REGION Network 33: RINSE-2_CLEANING_TIME_(PBFV-1,PBFV-17,PZDV-1,F-PUMP,PBFV-3,PBFV-4,PBFV-8,CIP-IN)
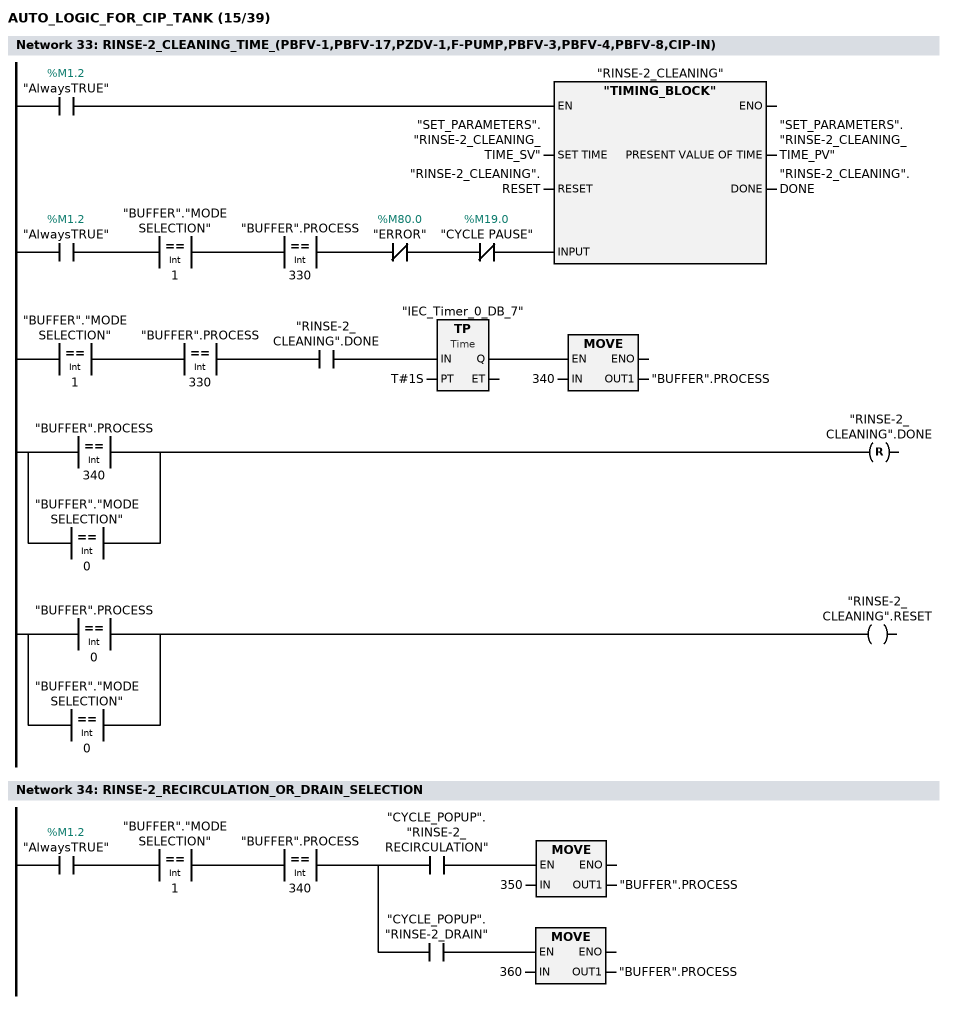
   RUNG wire#powerrail
      Contact( "AlwaysTRUE" )
      "RINSE-2_CLEANING"(INPUT := wire#w1, "SET TIME" := "SET_PARAMETERS"."RINSE-2_CLEANING_TIME_SV", RESET := "RINSE-2_CLEANING".RESET, "PRESENT VALUE OF TIME" => "SET_PARAMETERS"."RINSE-2_CLEANING_TIME_PV", DONE => "RINSE-2_CLEANING".DONE)
   END_RUNG
   RUNG wire#powerrail
      Contact( "AlwaysTRUE" )
      { S7_Templates := "SrcType := Int" } EQ_Contact(in1 := "BUFFER"."MODE SELECTION", in2 := 1)
      { S7_Templates := "SrcType := Int" } EQ_Contact(in1 := "BUFFER".PROCESS, in2 := 330)
      I_Contact( "ERROR" )
      I_Contact( "CYCLE PAUSE" )
   END_RUNG wire#w1
   RUNG wire#powerrail
      { S7_Templates := "SrcType := Int" } EQ_Contact(in1 := "BUFFER"."MODE SELECTION", in2 := 1)
      { S7_Templates := "SrcType := Int" } EQ_Contact(in1 := "BUFFER".PROCESS, in2 := 330)
      Contact( "RINSE-2_CLEANING".DONE )
      { S7_Templates := "time_type := Time" } "IEC_Timer_0_DB_7".TP(pt := T#1S, et =>)
      Move(in := 340, out1 => "BUFFER".PROCESS)
   END_RUNG
   RUNG wire#powerrail
      { S7_Templates := "SrcType := Int" } EQ_Contact(in1 := "BUFFER".PROCESS, in2 := 340)
      wire#w2
      R_Coil( "RINSE-2_CLEANING".DONE )
   END_RUNG
   RUNG wire#powerrail
      { S7_Templates := "SrcType := Int" } EQ_Contact(in1 := "BUFFER"."MODE SELECTION", in2 := 0)
   END_RUNG wire#w2
   RUNG wire#powerrail
      { S7_Templates := "SrcType := Int" } EQ_Contact(in1 := "BUFFER".PROCESS, in2 := 0)
      wire#w3
      Coil( "RINSE-2_CLEANING".RESET )
   END_RUNG
   RUNG wire#powerrail
      { S7_Templates := "SrcType := Int" } EQ_Contact(in1 := "BUFFER"."MODE SELECTION", in2 := 0)
   END_RUNG wire#w3
   // the same network as SCL:
   IF "AlwaysTRUE" THEN
       "RINSE-2_CLEANING"("SET TIME" := "SET_PARAMETERS"."RINSE-2_CLEANING_TIME_SV",   // "TIMING_BLOCK"
                          RESET := "RINSE-2_CLEANING".RESET,
                          INPUT := "AlwaysTRUE" AND ("BUFFER"."MODE SELECTION" = 1) AND ("BUFFER".PROCESS = 330) AND NOT "ERROR" AND NOT "CYCLE PAUSE",
                          "PRESENT VALUE OF TIME" => "SET_PARAMETERS"."RINSE-2_CLEANING_TIME_PV",
                          DONE => "RINSE-2_CLEANING".DONE);
   END_IF;
   "IEC_Timer_0_DB_7".TP(IN := ("BUFFER"."MODE SELECTION" = 1) AND ("BUFFER".PROCESS = 330) AND "RINSE-2_CLEANING".DONE,
                         PT := T#1S);
   IF "IEC_Timer_0_DB_7".Q THEN "BUFFER".PROCESS := 340; END_IF;
   IF ("BUFFER".PROCESS = 340) OR ("BUFFER"."MODE SELECTION" = 0) THEN
       "RINSE-2_CLEANING".DONE := FALSE;
   END_IF;
   "RINSE-2_CLEANING".RESET := ("BUFFER".PROCESS = 0) OR ("BUFFER"."MODE SELECTION" = 0);
END_REGION

REGION Network 34: RINSE-2_RECIRCULATION_OR_DRAIN_SELECTION
   RUNG wire#powerrail
      Contact( "AlwaysTRUE" )
      { S7_Templates := "SrcType := Int" } EQ_Contact(in1 := "BUFFER"."MODE SELECTION", in2 := 1)
      { S7_Templates := "SrcType := Int" } EQ_Contact(in1 := "BUFFER".PROCESS, in2 := 340)
      wire#w1
      Contact( "CYCLE_POPUP"."RINSE-2_RECIRCULATION" )
      Move(in := 350, out1 => "BUFFER".PROCESS)
   END_RUNG
   RUNG wire#w1
      Contact( "CYCLE_POPUP"."RINSE-2_DRAIN" )
      Move(in := 360, out1 => "BUFFER".PROCESS)
   END_RUNG
   // the same network as SCL:
   #_w1 := "AlwaysTRUE" AND ("BUFFER"."MODE SELECTION" = 1) AND ("BUFFER".PROCESS = 340);
   IF #_w1 AND "CYCLE_POPUP"."RINSE-2_RECIRCULATION" THEN "BUFFER".PROCESS := 350; END_IF;
   IF #_w1 AND "CYCLE_POPUP"."RINSE-2_DRAIN" THEN "BUFFER".PROCESS := 360; END_IF;
END_REGION

REGION Network 35: RINSE-2_RECIRCULATION_TIME_(CIP-OUT,R-PUMP,PBFV-6,PBFV-8,CIP-IN)
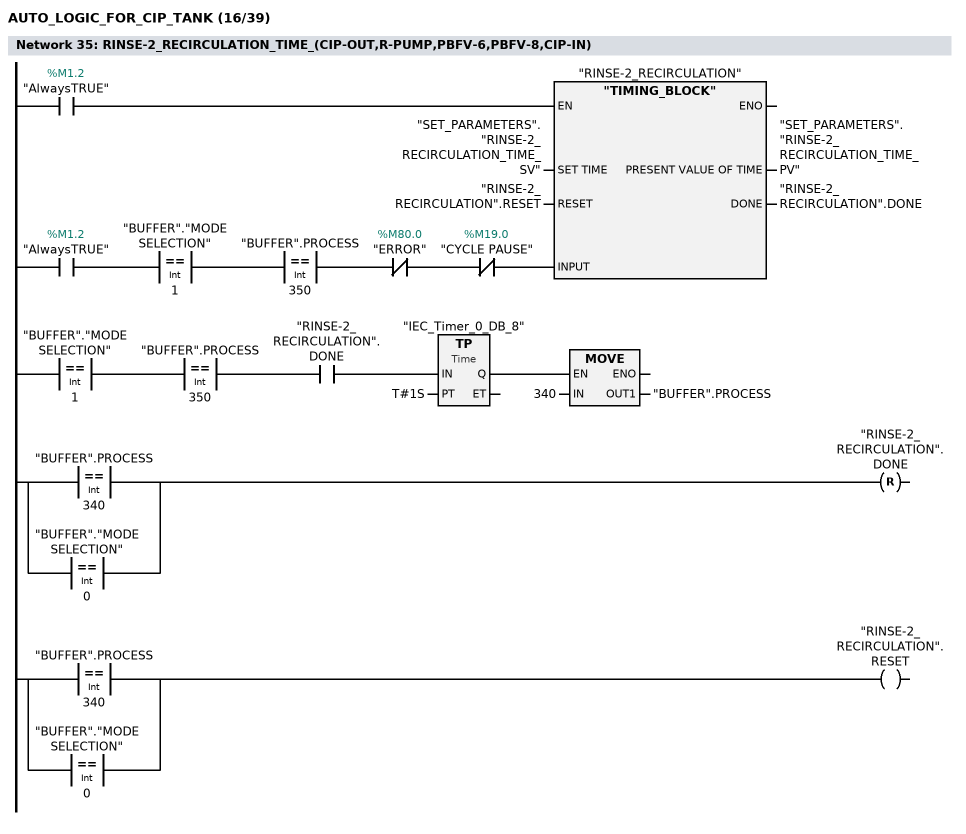
   RUNG wire#powerrail
      Contact( "AlwaysTRUE" )
      "RINSE-2_RECIRCULATION"(INPUT := wire#w1, "SET TIME" := "SET_PARAMETERS"."RINSE-2_RECIRCULATION_TIME_SV", RESET := "RINSE-2_RECIRCULATION".RESET, "PRESENT VALUE OF TIME" => "SET_PARAMETERS"."RINSE-2_RECIRCULATION_TIME_PV", DONE => "RINSE-2_RECIRCULATION".DONE)
   END_RUNG
   RUNG wire#powerrail
      Contact( "AlwaysTRUE" )
      { S7_Templates := "SrcType := Int" } EQ_Contact(in1 := "BUFFER"."MODE SELECTION", in2 := 1)
      { S7_Templates := "SrcType := Int" } EQ_Contact(in1 := "BUFFER".PROCESS, in2 := 350)
      I_Contact( "ERROR" )
      I_Contact( "CYCLE PAUSE" )
   END_RUNG wire#w1
   RUNG wire#powerrail
      { S7_Templates := "SrcType := Int" } EQ_Contact(in1 := "BUFFER"."MODE SELECTION", in2 := 1)
      { S7_Templates := "SrcType := Int" } EQ_Contact(in1 := "BUFFER".PROCESS, in2 := 350)
      Contact( "RINSE-2_RECIRCULATION".DONE )
      { S7_Templates := "time_type := Time" } "IEC_Timer_0_DB_8".TP(pt := T#1S, et =>)
      Move(in := 340, out1 => "BUFFER".PROCESS)
   END_RUNG
   RUNG wire#powerrail
      { S7_Templates := "SrcType := Int" } EQ_Contact(in1 := "BUFFER".PROCESS, in2 := 340)
      wire#w2
      R_Coil( "RINSE-2_RECIRCULATION".DONE )
   END_RUNG
   RUNG wire#powerrail
      { S7_Templates := "SrcType := Int" } EQ_Contact(in1 := "BUFFER"."MODE SELECTION", in2 := 0)
   END_RUNG wire#w2
   RUNG wire#powerrail
      { S7_Templates := "SrcType := Int" } EQ_Contact(in1 := "BUFFER".PROCESS, in2 := 340)
      wire#w3
      Coil( "RINSE-2_RECIRCULATION".RESET )
   END_RUNG
   RUNG wire#powerrail
      { S7_Templates := "SrcType := Int" } EQ_Contact(in1 := "BUFFER"."MODE SELECTION", in2 := 0)
   END_RUNG wire#w3
   // the same network as SCL:
   IF "AlwaysTRUE" THEN
       "RINSE-2_RECIRCULATION"("SET TIME" := "SET_PARAMETERS"."RINSE-2_RECIRCULATION_TIME_SV",   // "TIMING_BLOCK"
                               RESET := "RINSE-2_RECIRCULATION".RESET,
                               INPUT := "AlwaysTRUE" AND ("BUFFER"."MODE SELECTION" = 1) AND ("BUFFER".PROCESS = 350) AND NOT "ERROR" AND NOT "CYCLE PAUSE",
                               "PRESENT VALUE OF TIME" => "SET_PARAMETERS"."RINSE-2_RECIRCULATION_TIME_PV",
                               DONE => "RINSE-2_RECIRCULATION".DONE);
   END_IF;
   "IEC_Timer_0_DB_8".TP(IN := ("BUFFER"."MODE SELECTION" = 1) AND ("BUFFER".PROCESS = 350) AND "RINSE-2_RECIRCULATION".DONE,
                         PT := T#1S);
   IF "IEC_Timer_0_DB_8".Q THEN "BUFFER".PROCESS := 340; END_IF;
   IF ("BUFFER".PROCESS = 340) OR ("BUFFER"."MODE SELECTION" = 0) THEN
       "RINSE-2_RECIRCULATION".DONE := FALSE;
   END_IF;
   "RINSE-2_RECIRCULATION".RESET := ("BUFFER".PROCESS = 340) OR ("BUFFER"."MODE SELECTION" = 0);
END_REGION

REGION Network 36: RINSE-2_DRAIN_TIME_(CIP-OUT,R_PUMP,PBFV-11)
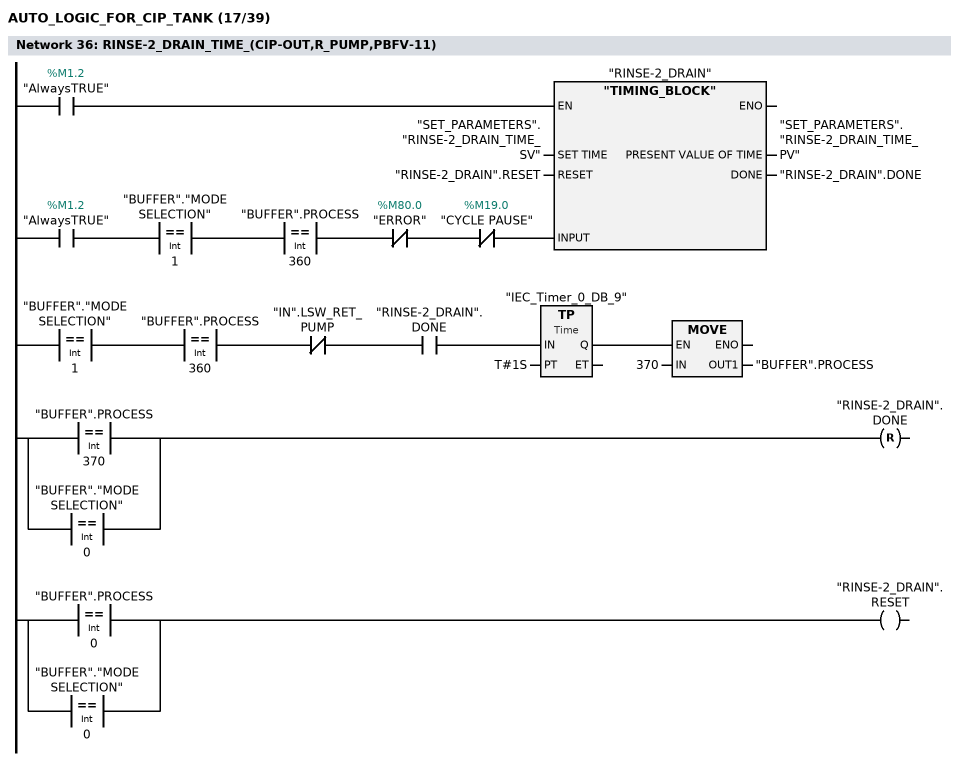
   RUNG wire#powerrail
      Contact( "AlwaysTRUE" )
      "RINSE-2_DRAIN"(INPUT := wire#w1, "SET TIME" := "SET_PARAMETERS"."RINSE-2_DRAIN_TIME_SV", RESET := "RINSE-2_DRAIN".RESET, "PRESENT VALUE OF TIME" => "SET_PARAMETERS"."RINSE-2_DRAIN_TIME_PV", DONE => "RINSE-2_DRAIN".DONE)
   END_RUNG
   RUNG wire#powerrail
      Contact( "AlwaysTRUE" )
      { S7_Templates := "SrcType := Int" } EQ_Contact(in1 := "BUFFER"."MODE SELECTION", in2 := 1)
      { S7_Templates := "SrcType := Int" } EQ_Contact(in1 := "BUFFER".PROCESS, in2 := 360)
      I_Contact( "ERROR" )
      I_Contact( "CYCLE PAUSE" )
   END_RUNG wire#w1
   RUNG wire#powerrail
      { S7_Templates := "SrcType := Int" } EQ_Contact(in1 := "BUFFER"."MODE SELECTION", in2 := 1)
      { S7_Templates := "SrcType := Int" } EQ_Contact(in1 := "BUFFER".PROCESS, in2 := 360)
      I_Contact( "IN".LSW_RET_PUMP )
      Contact( "RINSE-2_DRAIN".DONE )
      { S7_Templates := "time_type := Time" } "IEC_Timer_0_DB_9".TP(pt := T#1S, et =>)
      Move(in := 370, out1 => "BUFFER".PROCESS)
   END_RUNG
   RUNG wire#powerrail
      { S7_Templates := "SrcType := Int" } EQ_Contact(in1 := "BUFFER".PROCESS, in2 := 370)
      wire#w2
      R_Coil( "RINSE-2_DRAIN".DONE )
   END_RUNG
   RUNG wire#powerrail
      { S7_Templates := "SrcType := Int" } EQ_Contact(in1 := "BUFFER"."MODE SELECTION", in2 := 0)
   END_RUNG wire#w2
   RUNG wire#powerrail
      { S7_Templates := "SrcType := Int" } EQ_Contact(in1 := "BUFFER".PROCESS, in2 := 0)
      wire#w3
      Coil( "RINSE-2_DRAIN".RESET )
   END_RUNG
   RUNG wire#powerrail
      { S7_Templates := "SrcType := Int" } EQ_Contact(in1 := "BUFFER"."MODE SELECTION", in2 := 0)
   END_RUNG wire#w3
   // the same network as SCL:
   IF "AlwaysTRUE" THEN
       "RINSE-2_DRAIN"("SET TIME" := "SET_PARAMETERS"."RINSE-2_DRAIN_TIME_SV",   // "TIMING_BLOCK"
                       RESET := "RINSE-2_DRAIN".RESET,
                       INPUT := "AlwaysTRUE" AND ("BUFFER"."MODE SELECTION" = 1) AND ("BUFFER".PROCESS = 360) AND NOT "ERROR" AND NOT "CYCLE PAUSE",
                       "PRESENT VALUE OF TIME" => "SET_PARAMETERS"."RINSE-2_DRAIN_TIME_PV",
                       DONE => "RINSE-2_DRAIN".DONE);
   END_IF;
   "IEC_Timer_0_DB_9".TP(IN := ("BUFFER"."MODE SELECTION" = 1) AND ("BUFFER".PROCESS = 360) AND NOT "IN".LSW_RET_PUMP AND "RINSE-2_DRAIN".DONE,
                         PT := T#1S);
   IF "IEC_Timer_0_DB_9".Q THEN "BUFFER".PROCESS := 370; END_IF;
   IF ("BUFFER".PROCESS = 370) OR ("BUFFER"."MODE SELECTION" = 0) THEN "RINSE-2_DRAIN".DONE := FALSE; END_IF;
   "RINSE-2_DRAIN".RESET := ("BUFFER".PROCESS = 0) OR ("BUFFER"."MODE SELECTION" = 0);
END_REGION

REGION Network 37: RINSE-2_PUMP_CHASING_TIME_(PBFV-12,PBFV13)
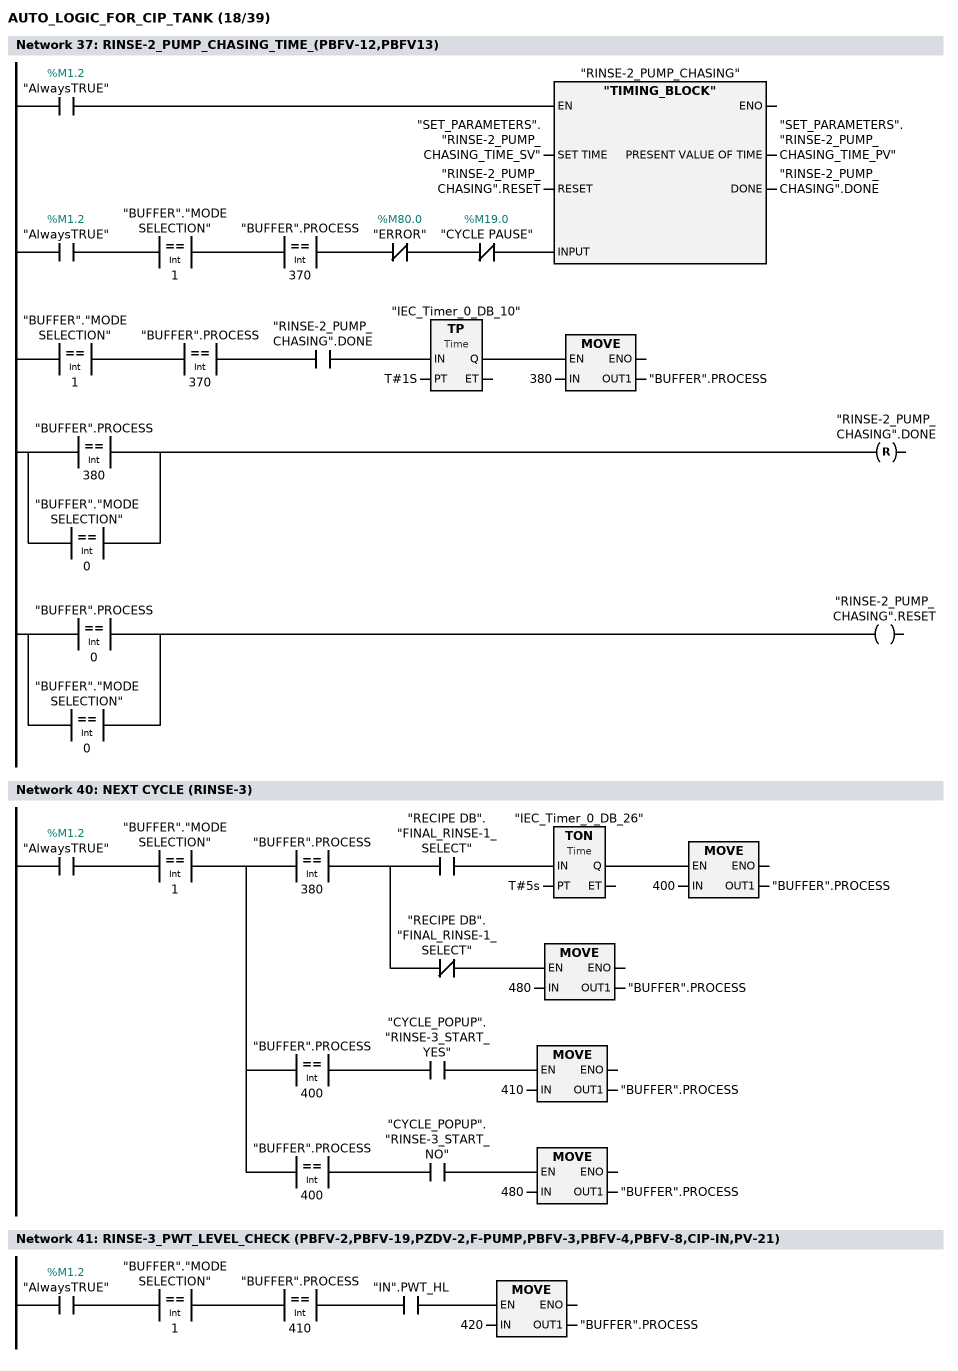
   RUNG wire#powerrail
      Contact( "AlwaysTRUE" )
      "RINSE-2_PUMP_CHASING"(INPUT := wire#w1, "SET TIME" := "SET_PARAMETERS"."RINSE-2_PUMP_CHASING_TIME_SV", RESET := "RINSE-2_PUMP_CHASING".RESET, "PRESENT VALUE OF TIME" => "SET_PARAMETERS"."RINSE-2_PUMP_CHASING_TIME_PV", DONE => "RINSE-2_PUMP_CHASING".DONE)
   END_RUNG
   RUNG wire#powerrail
      Contact( "AlwaysTRUE" )
      { S7_Templates := "SrcType := Int" } EQ_Contact(in1 := "BUFFER"."MODE SELECTION", in2 := 1)
      { S7_Templates := "SrcType := Int" } EQ_Contact(in1 := "BUFFER".PROCESS, in2 := 370)
      I_Contact( "ERROR" )
      I_Contact( "CYCLE PAUSE" )
   END_RUNG wire#w1
   RUNG wire#powerrail
      { S7_Templates := "SrcType := Int" } EQ_Contact(in1 := "BUFFER"."MODE SELECTION", in2 := 1)
      { S7_Templates := "SrcType := Int" } EQ_Contact(in1 := "BUFFER".PROCESS, in2 := 370)
      Contact( "RINSE-2_PUMP_CHASING".DONE )
      { S7_Templates := "time_type := Time" } "IEC_Timer_0_DB_10".TP(pt := T#1S, et =>)
      Move(in := 380, out1 => "BUFFER".PROCESS)
   END_RUNG
   RUNG wire#powerrail
      { S7_Templates := "SrcType := Int" } EQ_Contact(in1 := "BUFFER".PROCESS, in2 := 380)
      wire#w2
      R_Coil( "RINSE-2_PUMP_CHASING".DONE )
   END_RUNG
   RUNG wire#powerrail
      { S7_Templates := "SrcType := Int" } EQ_Contact(in1 := "BUFFER"."MODE SELECTION", in2 := 0)
   END_RUNG wire#w2
   RUNG wire#powerrail
      { S7_Templates := "SrcType := Int" } EQ_Contact(in1 := "BUFFER".PROCESS, in2 := 0)
      wire#w3
      Coil( "RINSE-2_PUMP_CHASING".RESET )
   END_RUNG
   RUNG wire#powerrail
      { S7_Templates := "SrcType := Int" } EQ_Contact(in1 := "BUFFER"."MODE SELECTION", in2 := 0)
   END_RUNG wire#w3
   // the same network as SCL:
   IF "AlwaysTRUE" THEN
       "RINSE-2_PUMP_CHASING"("SET TIME" := "SET_PARAMETERS"."RINSE-2_PUMP_CHASING_TIME_SV",   // "TIMING_BLOCK"
                              RESET := "RINSE-2_PUMP_CHASING".RESET,
                              INPUT := "AlwaysTRUE" AND ("BUFFER"."MODE SELECTION" = 1) AND ("BUFFER".PROCESS = 370) AND NOT "ERROR" AND NOT "CYCLE PAUSE",
                              "PRESENT VALUE OF TIME" => "SET_PARAMETERS"."RINSE-2_PUMP_CHASING_TIME_PV",
                              DONE => "RINSE-2_PUMP_CHASING".DONE);
   END_IF;
   "IEC_Timer_0_DB_10".TP(IN := ("BUFFER"."MODE SELECTION" = 1) AND ("BUFFER".PROCESS = 370) AND "RINSE-2_PUMP_CHASING".DONE,
                          PT := T#1S);
   IF "IEC_Timer_0_DB_10".Q THEN "BUFFER".PROCESS := 380; END_IF;
   IF ("BUFFER".PROCESS = 380) OR ("BUFFER"."MODE SELECTION" = 0) THEN
       "RINSE-2_PUMP_CHASING".DONE := FALSE;
   END_IF;
   "RINSE-2_PUMP_CHASING".RESET := ("BUFFER".PROCESS = 0) OR ("BUFFER"."MODE SELECTION" = 0);
END_REGION

REGION Network 40: NEXT CYCLE (RINSE-3)
   RUNG wire#powerrail
      Contact( "AlwaysTRUE" )
      { S7_Templates := "SrcType := Int" } EQ_Contact(in1 := "BUFFER"."MODE SELECTION", in2 := 1)
      wire#w1
      { S7_Templates := "SrcType := Int" } EQ_Contact(in1 := "BUFFER".PROCESS, in2 := 380)
      wire#w2
      Contact( "RECIPE DB"."FINAL_RINSE-1_SELECT" )
      { S7_Templates := "time_type := Time" } "IEC_Timer_0_DB_26".TON(pt := T#5s, et =>)
      Move(in := 400, out1 => "BUFFER".PROCESS)
   END_RUNG
   RUNG wire#w2
      I_Contact( "RECIPE DB"."FINAL_RINSE-1_SELECT" )
      Move(in := 480, out1 => "BUFFER".PROCESS)
   END_RUNG
   RUNG wire#w1
      { S7_Templates := "SrcType := Int" } EQ_Contact(in1 := "BUFFER".PROCESS, in2 := 400)
      Contact( "CYCLE_POPUP"."RINSE-3_START_YES" )
      Move(in := 410, out1 => "BUFFER".PROCESS)
   END_RUNG
   RUNG wire#w1
      { S7_Templates := "SrcType := Int" } EQ_Contact(in1 := "BUFFER".PROCESS, in2 := 400)
      Contact( "CYCLE_POPUP"."RINSE-3_START_NO" )
      Move(in := 480, out1 => "BUFFER".PROCESS)
   END_RUNG
   // the same network as SCL:
   #_w1 := "AlwaysTRUE" AND ("BUFFER"."MODE SELECTION" = 1);
   #_w2 := #_w1 AND ("BUFFER".PROCESS = 380);
   "IEC_Timer_0_DB_26".TON(IN := #_w2 AND "RECIPE DB"."FINAL_RINSE-1_SELECT", PT := T#5s);
   IF "IEC_Timer_0_DB_26".Q THEN "BUFFER".PROCESS := 400; END_IF;
   IF #_w2 AND NOT "RECIPE DB"."FINAL_RINSE-1_SELECT" THEN "BUFFER".PROCESS := 480; END_IF;
   IF #_w1 AND ("BUFFER".PROCESS = 400) AND "CYCLE_POPUP"."RINSE-3_START_YES" THEN
       "BUFFER".PROCESS := 410;
   END_IF;
   IF #_w1 AND ("BUFFER".PROCESS = 400) AND "CYCLE_POPUP"."RINSE-3_START_NO" THEN
       "BUFFER".PROCESS := 480;
   END_IF;
END_REGION

REGION Network 41: RINSE-3_PWT_LEVEL_CHECK (PBFV-2,PBFV-19,PZDV-2,F-PUMP,PBFV-3,PBFV-4,PBFV-8,CIP-IN,PV-21)
   RUNG wire#powerrail
      Contact( "AlwaysTRUE" )
      { S7_Templates := "SrcType := Int" } EQ_Contact(in1 := "BUFFER"."MODE SELECTION", in2 := 1)
      { S7_Templates := "SrcType := Int" } EQ_Contact(in1 := "BUFFER".PROCESS, in2 := 410)
      Contact( "IN".PWT_HL )
      Move(in := 420, out1 => "BUFFER".PROCESS)
   END_RUNG
   // the same network as SCL:
   IF "AlwaysTRUE" AND ("BUFFER"."MODE SELECTION" = 1) AND ("BUFFER".PROCESS = 410) AND "IN".PWT_HL THEN
       "BUFFER".PROCESS := 420;
   END_IF;
END_REGION

REGION Network 42: RINSE-3_TEMP_CHECK _(PBFV-2,PBFV-19,PZDV-2,F-PUMP,PBFV-3,PBFV-4,PBFV-8,CIP-IN)
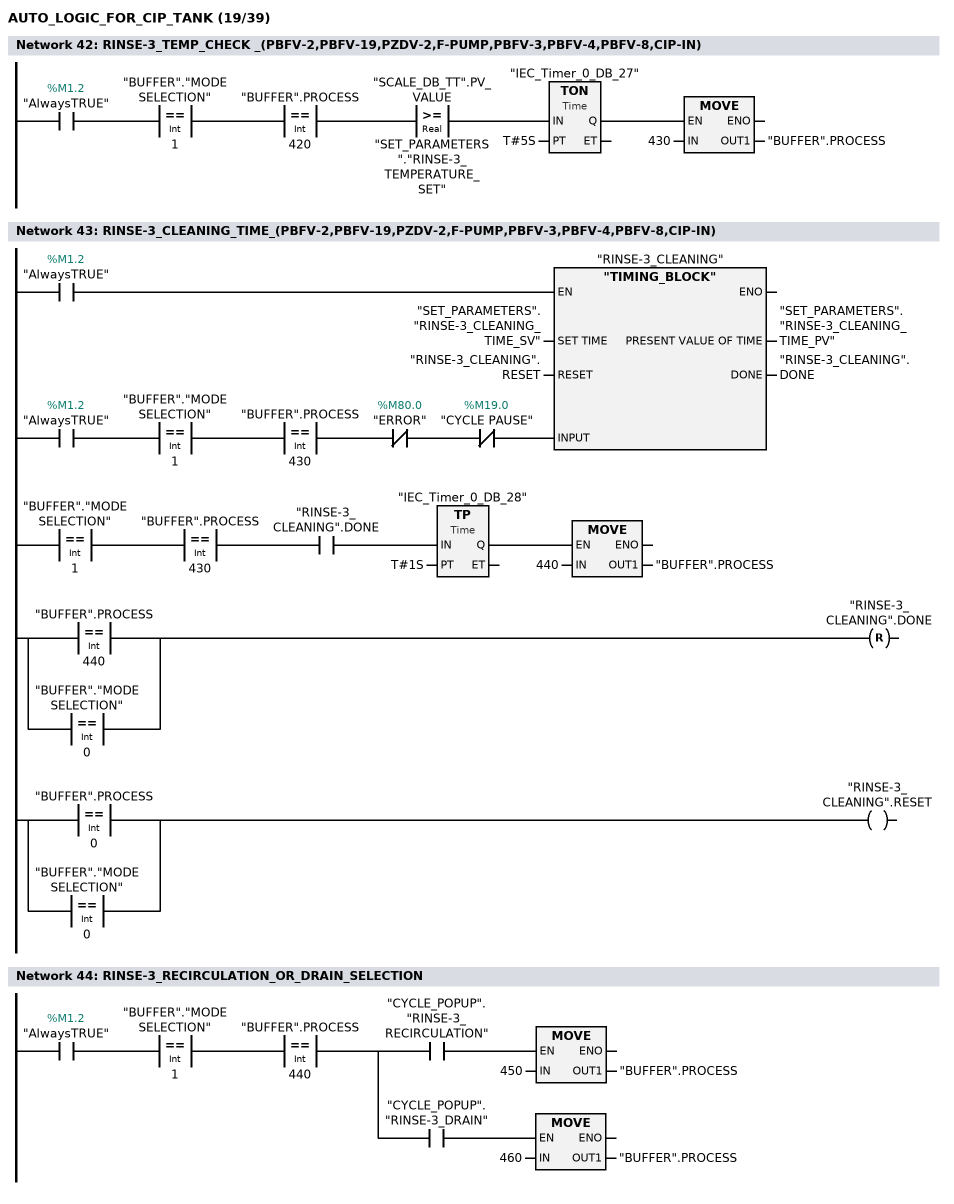
   RUNG wire#powerrail
      Contact( "AlwaysTRUE" )
      { S7_Templates := "SrcType := Int" } EQ_Contact(in1 := "BUFFER"."MODE SELECTION", in2 := 1)
      { S7_Templates := "SrcType := Int" } EQ_Contact(in1 := "BUFFER".PROCESS, in2 := 420)
      { S7_Templates := "SrcType := Real" } GE_Contact(in1 := "SCALE_DB_TT".PV_VALUE, in2 := "SET_PARAMETERS"."RINSE-3_TEMPERATURE_SET")
      { S7_Templates := "time_type := Time" } "IEC_Timer_0_DB_27".TON(pt := T#5S, et =>)
      Move(in := 430, out1 => "BUFFER".PROCESS)
   END_RUNG
   // the same network as SCL:
   "IEC_Timer_0_DB_27".TON(IN := "AlwaysTRUE" AND ("BUFFER"."MODE SELECTION" = 1) AND ("BUFFER".PROCESS = 420) AND ("SCALE_DB_TT".PV_VALUE >= "SET_PARAMETERS"."RINSE-3_TEMPERATURE_SET"),
                           PT := T#5S);
   IF "IEC_Timer_0_DB_27".Q THEN "BUFFER".PROCESS := 430; END_IF;
END_REGION

REGION Network 43: RINSE-3_CLEANING_TIME_(PBFV-2,PBFV-19,PZDV-2,F-PUMP,PBFV-3,PBFV-4,PBFV-8,CIP-IN)
   RUNG wire#powerrail
      Contact( "AlwaysTRUE" )
      "RINSE-3_CLEANING"(INPUT := wire#w1, "SET TIME" := "SET_PARAMETERS"."RINSE-3_CLEANING_TIME_SV", RESET := "RINSE-3_CLEANING".RESET, "PRESENT VALUE OF TIME" => "SET_PARAMETERS"."RINSE-3_CLEANING_TIME_PV", DONE => "RINSE-3_CLEANING".DONE)
   END_RUNG
   RUNG wire#powerrail
      Contact( "AlwaysTRUE" )
      { S7_Templates := "SrcType := Int" } EQ_Contact(in1 := "BUFFER"."MODE SELECTION", in2 := 1)
      { S7_Templates := "SrcType := Int" } EQ_Contact(in1 := "BUFFER".PROCESS, in2 := 430)
      I_Contact( "ERROR" )
      I_Contact( "CYCLE PAUSE" )
   END_RUNG wire#w1
   RUNG wire#powerrail
      { S7_Templates := "SrcType := Int" } EQ_Contact(in1 := "BUFFER"."MODE SELECTION", in2 := 1)
      { S7_Templates := "SrcType := Int" } EQ_Contact(in1 := "BUFFER".PROCESS, in2 := 430)
      Contact( "RINSE-3_CLEANING".DONE )
      { S7_Templates := "time_type := Time" } "IEC_Timer_0_DB_28".TP(pt := T#1S, et =>)
      Move(in := 440, out1 => "BUFFER".PROCESS)
   END_RUNG
   RUNG wire#powerrail
      { S7_Templates := "SrcType := Int" } EQ_Contact(in1 := "BUFFER".PROCESS, in2 := 440)
      wire#w2
      R_Coil( "RINSE-3_CLEANING".DONE )
   END_RUNG
   RUNG wire#powerrail
      { S7_Templates := "SrcType := Int" } EQ_Contact(in1 := "BUFFER"."MODE SELECTION", in2 := 0)
   END_RUNG wire#w2
   RUNG wire#powerrail
      { S7_Templates := "SrcType := Int" } EQ_Contact(in1 := "BUFFER".PROCESS, in2 := 0)
      wire#w3
      Coil( "RINSE-3_CLEANING".RESET )
   END_RUNG
   RUNG wire#powerrail
      { S7_Templates := "SrcType := Int" } EQ_Contact(in1 := "BUFFER"."MODE SELECTION", in2 := 0)
   END_RUNG wire#w3
   // the same network as SCL:
   IF "AlwaysTRUE" THEN
       "RINSE-3_CLEANING"("SET TIME" := "SET_PARAMETERS"."RINSE-3_CLEANING_TIME_SV",   // "TIMING_BLOCK"
                          RESET := "RINSE-3_CLEANING".RESET,
                          INPUT := "AlwaysTRUE" AND ("BUFFER"."MODE SELECTION" = 1) AND ("BUFFER".PROCESS = 430) AND NOT "ERROR" AND NOT "CYCLE PAUSE",
                          "PRESENT VALUE OF TIME" => "SET_PARAMETERS"."RINSE-3_CLEANING_TIME_PV",
                          DONE => "RINSE-3_CLEANING".DONE);
   END_IF;
   "IEC_Timer_0_DB_28".TP(IN := ("BUFFER"."MODE SELECTION" = 1) AND ("BUFFER".PROCESS = 430) AND "RINSE-3_CLEANING".DONE,
                          PT := T#1S);
   IF "IEC_Timer_0_DB_28".Q THEN "BUFFER".PROCESS := 440; END_IF;
   IF ("BUFFER".PROCESS = 440) OR ("BUFFER"."MODE SELECTION" = 0) THEN
       "RINSE-3_CLEANING".DONE := FALSE;
   END_IF;
   "RINSE-3_CLEANING".RESET := ("BUFFER".PROCESS = 0) OR ("BUFFER"."MODE SELECTION" = 0);
END_REGION

REGION Network 44: RINSE-3_RECIRCULATION_OR_DRAIN_SELECTION
   RUNG wire#powerrail
      Contact( "AlwaysTRUE" )
      { S7_Templates := "SrcType := Int" } EQ_Contact(in1 := "BUFFER"."MODE SELECTION", in2 := 1)
      { S7_Templates := "SrcType := Int" } EQ_Contact(in1 := "BUFFER".PROCESS, in2 := 440)
      wire#w1
      Contact( "CYCLE_POPUP"."RINSE-3_RECIRCULATION" )
      Move(in := 450, out1 => "BUFFER".PROCESS)
   END_RUNG
   RUNG wire#w1
      Contact( "CYCLE_POPUP"."RINSE-3_DRAIN" )
      Move(in := 460, out1 => "BUFFER".PROCESS)
   END_RUNG
   // the same network as SCL:
   #_w1 := "AlwaysTRUE" AND ("BUFFER"."MODE SELECTION" = 1) AND ("BUFFER".PROCESS = 440);
   IF #_w1 AND "CYCLE_POPUP"."RINSE-3_RECIRCULATION" THEN "BUFFER".PROCESS := 450; END_IF;
   IF #_w1 AND "CYCLE_POPUP"."RINSE-3_DRAIN" THEN "BUFFER".PROCESS := 460; END_IF;
END_REGION

REGION Network 45: RINSE-3_RECIRCULATION_TIME_(CIP-OUT,R-PUMP,PBFV-6,PBFV-8,CIP-IN)
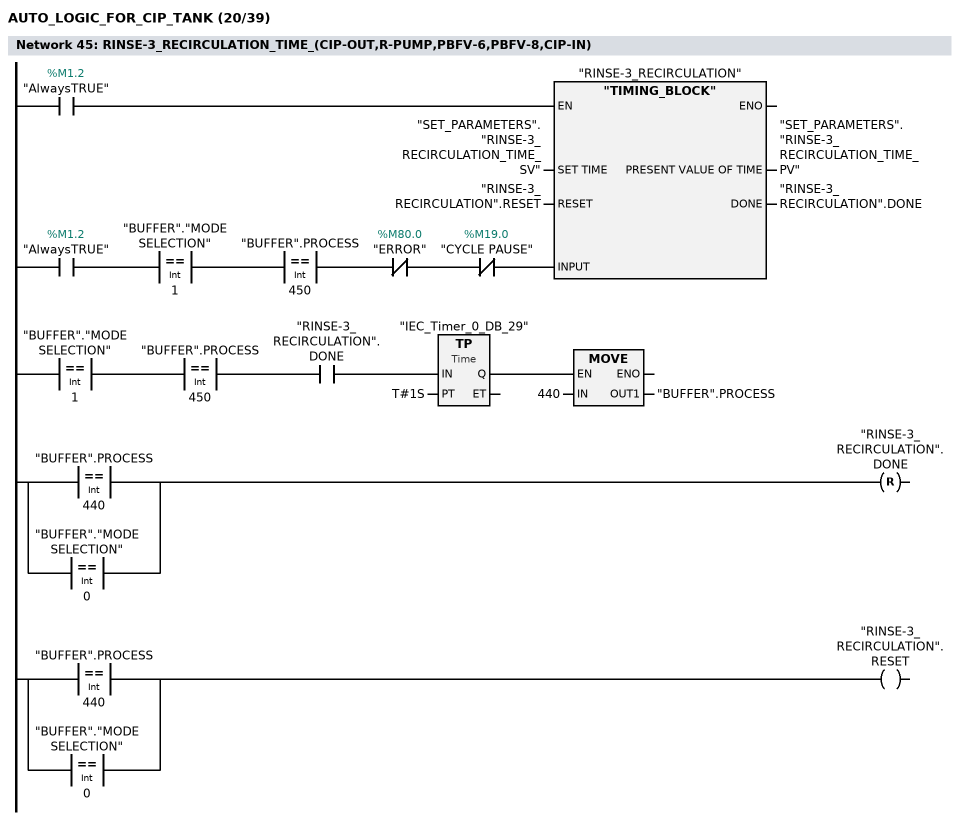
   RUNG wire#powerrail
      Contact( "AlwaysTRUE" )
      "RINSE-3_RECIRCULATION"(INPUT := wire#w1, "SET TIME" := "SET_PARAMETERS"."RINSE-3_RECIRCULATION_TIME_SV", RESET := "RINSE-3_RECIRCULATION".RESET, "PRESENT VALUE OF TIME" => "SET_PARAMETERS"."RINSE-3_RECIRCULATION_TIME_PV", DONE => "RINSE-3_RECIRCULATION".DONE)
   END_RUNG
   RUNG wire#powerrail
      Contact( "AlwaysTRUE" )
      { S7_Templates := "SrcType := Int" } EQ_Contact(in1 := "BUFFER"."MODE SELECTION", in2 := 1)
      { S7_Templates := "SrcType := Int" } EQ_Contact(in1 := "BUFFER".PROCESS, in2 := 450)
      I_Contact( "ERROR" )
      I_Contact( "CYCLE PAUSE" )
   END_RUNG wire#w1
   RUNG wire#powerrail
      { S7_Templates := "SrcType := Int" } EQ_Contact(in1 := "BUFFER"."MODE SELECTION", in2 := 1)
      { S7_Templates := "SrcType := Int" } EQ_Contact(in1 := "BUFFER".PROCESS, in2 := 450)
      Contact( "RINSE-3_RECIRCULATION".DONE )
      { S7_Templates := "time_type := Time" } "IEC_Timer_0_DB_29".TP(pt := T#1S, et =>)
      Move(in := 440, out1 => "BUFFER".PROCESS)
   END_RUNG
   RUNG wire#powerrail
      { S7_Templates := "SrcType := Int" } EQ_Contact(in1 := "BUFFER".PROCESS, in2 := 440)
      wire#w2
      R_Coil( "RINSE-3_RECIRCULATION".DONE )
   END_RUNG
   RUNG wire#powerrail
      { S7_Templates := "SrcType := Int" } EQ_Contact(in1 := "BUFFER"."MODE SELECTION", in2 := 0)
   END_RUNG wire#w2
   RUNG wire#powerrail
      { S7_Templates := "SrcType := Int" } EQ_Contact(in1 := "BUFFER".PROCESS, in2 := 440)
      wire#w3
      Coil( "RINSE-3_RECIRCULATION".RESET )
   END_RUNG
   RUNG wire#powerrail
      { S7_Templates := "SrcType := Int" } EQ_Contact(in1 := "BUFFER"."MODE SELECTION", in2 := 0)
   END_RUNG wire#w3
   // the same network as SCL:
   IF "AlwaysTRUE" THEN
       "RINSE-3_RECIRCULATION"("SET TIME" := "SET_PARAMETERS"."RINSE-3_RECIRCULATION_TIME_SV",   // "TIMING_BLOCK"
                               RESET := "RINSE-3_RECIRCULATION".RESET,
                               INPUT := "AlwaysTRUE" AND ("BUFFER"."MODE SELECTION" = 1) AND ("BUFFER".PROCESS = 450) AND NOT "ERROR" AND NOT "CYCLE PAUSE",
                               "PRESENT VALUE OF TIME" => "SET_PARAMETERS"."RINSE-3_RECIRCULATION_TIME_PV",
                               DONE => "RINSE-3_RECIRCULATION".DONE);
   END_IF;
   "IEC_Timer_0_DB_29".TP(IN := ("BUFFER"."MODE SELECTION" = 1) AND ("BUFFER".PROCESS = 450) AND "RINSE-3_RECIRCULATION".DONE,
                          PT := T#1S);
   IF "IEC_Timer_0_DB_29".Q THEN "BUFFER".PROCESS := 440; END_IF;
   IF ("BUFFER".PROCESS = 440) OR ("BUFFER"."MODE SELECTION" = 0) THEN
       "RINSE-3_RECIRCULATION".DONE := FALSE;
   END_IF;
   "RINSE-3_RECIRCULATION".RESET := ("BUFFER".PROCESS = 440) OR ("BUFFER"."MODE SELECTION" = 0);
END_REGION

REGION Network 46: RINSE-3_DRAIN_TIME_(CIP-OUT,R_PUMP,PBFV-11)
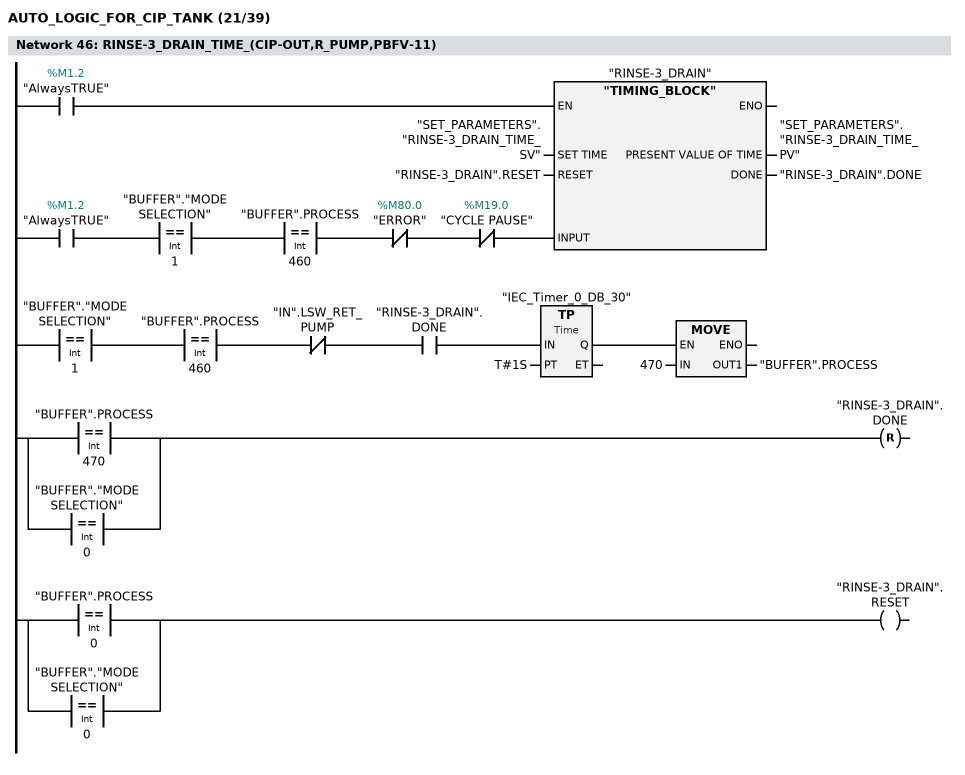
   RUNG wire#powerrail
      Contact( "AlwaysTRUE" )
      "RINSE-3_DRAIN"(INPUT := wire#w1, "SET TIME" := "SET_PARAMETERS"."RINSE-3_DRAIN_TIME_SV", RESET := "RINSE-3_DRAIN".RESET, "PRESENT VALUE OF TIME" => "SET_PARAMETERS"."RINSE-3_DRAIN_TIME_PV", DONE => "RINSE-3_DRAIN".DONE)
   END_RUNG
   RUNG wire#powerrail
      Contact( "AlwaysTRUE" )
      { S7_Templates := "SrcType := Int" } EQ_Contact(in1 := "BUFFER"."MODE SELECTION", in2 := 1)
      { S7_Templates := "SrcType := Int" } EQ_Contact(in1 := "BUFFER".PROCESS, in2 := 460)
      I_Contact( "ERROR" )
      I_Contact( "CYCLE PAUSE" )
   END_RUNG wire#w1
   RUNG wire#powerrail
      { S7_Templates := "SrcType := Int" } EQ_Contact(in1 := "BUFFER"."MODE SELECTION", in2 := 1)
      { S7_Templates := "SrcType := Int" } EQ_Contact(in1 := "BUFFER".PROCESS, in2 := 460)
      I_Contact( "IN".LSW_RET_PUMP )
      Contact( "RINSE-3_DRAIN".DONE )
      { S7_Templates := "time_type := Time" } "IEC_Timer_0_DB_30".TP(pt := T#1S, et =>)
      Move(in := 470, out1 => "BUFFER".PROCESS)
   END_RUNG
   RUNG wire#powerrail
      { S7_Templates := "SrcType := Int" } EQ_Contact(in1 := "BUFFER".PROCESS, in2 := 470)
      wire#w2
      R_Coil( "RINSE-3_DRAIN".DONE )
   END_RUNG
   RUNG wire#powerrail
      { S7_Templates := "SrcType := Int" } EQ_Contact(in1 := "BUFFER"."MODE SELECTION", in2 := 0)
   END_RUNG wire#w2
   RUNG wire#powerrail
      { S7_Templates := "SrcType := Int" } EQ_Contact(in1 := "BUFFER".PROCESS, in2 := 0)
      wire#w3
      Coil( "RINSE-3_DRAIN".RESET )
   END_RUNG
   RUNG wire#powerrail
      { S7_Templates := "SrcType := Int" } EQ_Contact(in1 := "BUFFER"."MODE SELECTION", in2 := 0)
   END_RUNG wire#w3
   // the same network as SCL:
   IF "AlwaysTRUE" THEN
       "RINSE-3_DRAIN"("SET TIME" := "SET_PARAMETERS"."RINSE-3_DRAIN_TIME_SV",   // "TIMING_BLOCK"
                       RESET := "RINSE-3_DRAIN".RESET,
                       INPUT := "AlwaysTRUE" AND ("BUFFER"."MODE SELECTION" = 1) AND ("BUFFER".PROCESS = 460) AND NOT "ERROR" AND NOT "CYCLE PAUSE",
                       "PRESENT VALUE OF TIME" => "SET_PARAMETERS"."RINSE-3_DRAIN_TIME_PV",
                       DONE => "RINSE-3_DRAIN".DONE);
   END_IF;
   "IEC_Timer_0_DB_30".TP(IN := ("BUFFER"."MODE SELECTION" = 1) AND ("BUFFER".PROCESS = 460) AND NOT "IN".LSW_RET_PUMP AND "RINSE-3_DRAIN".DONE,
                          PT := T#1S);
   IF "IEC_Timer_0_DB_30".Q THEN "BUFFER".PROCESS := 470; END_IF;
   IF ("BUFFER".PROCESS = 470) OR ("BUFFER"."MODE SELECTION" = 0) THEN "RINSE-3_DRAIN".DONE := FALSE; END_IF;
   "RINSE-3_DRAIN".RESET := ("BUFFER".PROCESS = 0) OR ("BUFFER"."MODE SELECTION" = 0);
END_REGION

REGION Network 47: RINSE-3_PUMP_CHASING_TIME_(PBFV-12,PBFV13)
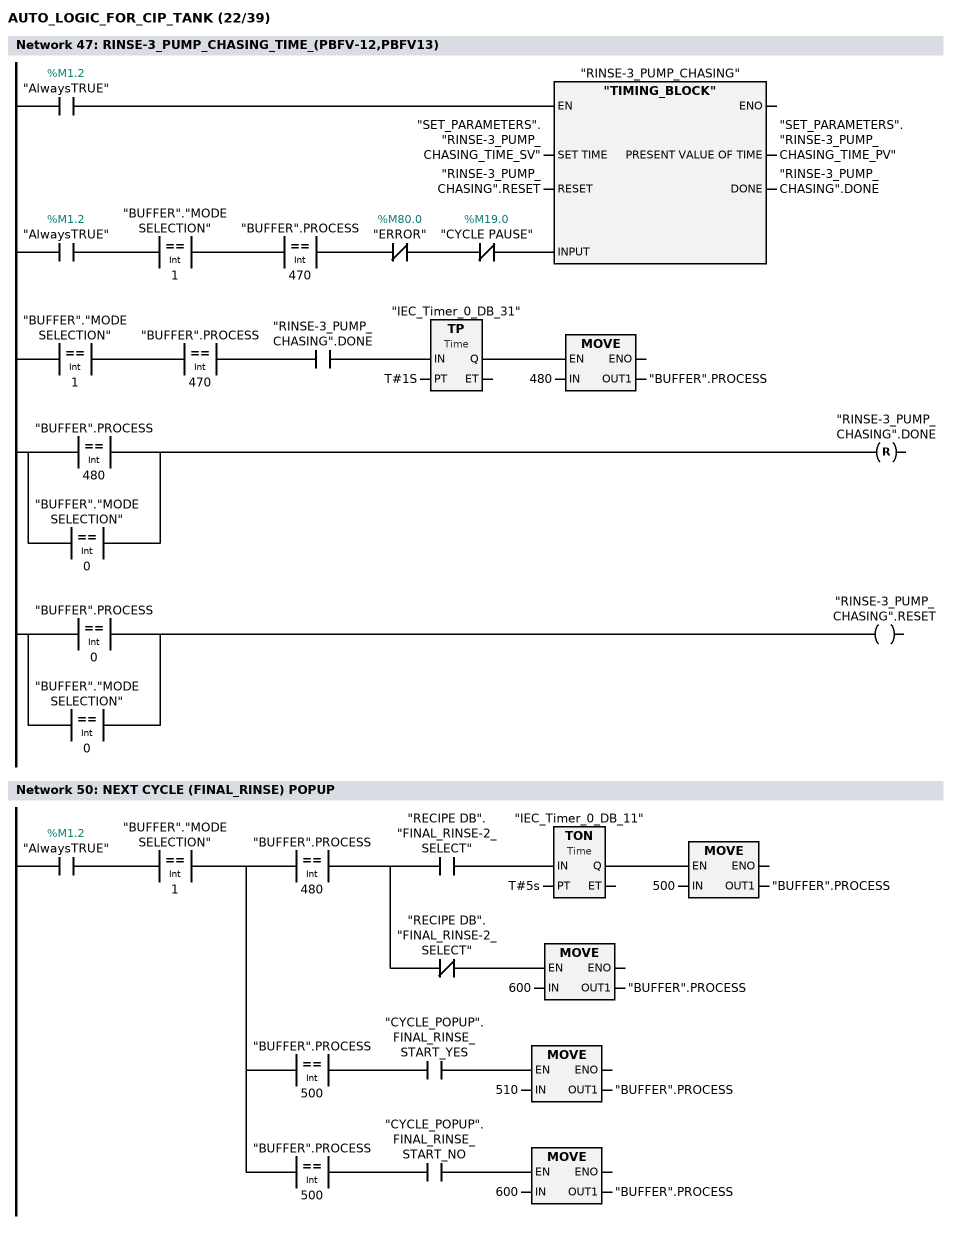
   RUNG wire#powerrail
      Contact( "AlwaysTRUE" )
      "RINSE-3_PUMP_CHASING"(INPUT := wire#w1, "SET TIME" := "SET_PARAMETERS"."RINSE-3_PUMP_CHASING_TIME_SV", RESET := "RINSE-3_PUMP_CHASING".RESET, "PRESENT VALUE OF TIME" => "SET_PARAMETERS"."RINSE-3_PUMP_CHASING_TIME_PV", DONE => "RINSE-3_PUMP_CHASING".DONE)
   END_RUNG
   RUNG wire#powerrail
      Contact( "AlwaysTRUE" )
      { S7_Templates := "SrcType := Int" } EQ_Contact(in1 := "BUFFER"."MODE SELECTION", in2 := 1)
      { S7_Templates := "SrcType := Int" } EQ_Contact(in1 := "BUFFER".PROCESS, in2 := 470)
      I_Contact( "ERROR" )
      I_Contact( "CYCLE PAUSE" )
   END_RUNG wire#w1
   RUNG wire#powerrail
      { S7_Templates := "SrcType := Int" } EQ_Contact(in1 := "BUFFER"."MODE SELECTION", in2 := 1)
      { S7_Templates := "SrcType := Int" } EQ_Contact(in1 := "BUFFER".PROCESS, in2 := 470)
      Contact( "RINSE-3_PUMP_CHASING".DONE )
      { S7_Templates := "time_type := Time" } "IEC_Timer_0_DB_31".TP(pt := T#1S, et =>)
      Move(in := 480, out1 => "BUFFER".PROCESS)
   END_RUNG
   RUNG wire#powerrail
      { S7_Templates := "SrcType := Int" } EQ_Contact(in1 := "BUFFER".PROCESS, in2 := 480)
      wire#w2
      R_Coil( "RINSE-3_PUMP_CHASING".DONE )
   END_RUNG
   RUNG wire#powerrail
      { S7_Templates := "SrcType := Int" } EQ_Contact(in1 := "BUFFER"."MODE SELECTION", in2 := 0)
   END_RUNG wire#w2
   RUNG wire#powerrail
      { S7_Templates := "SrcType := Int" } EQ_Contact(in1 := "BUFFER".PROCESS, in2 := 0)
      wire#w3
      Coil( "RINSE-3_PUMP_CHASING".RESET )
   END_RUNG
   RUNG wire#powerrail
      { S7_Templates := "SrcType := Int" } EQ_Contact(in1 := "BUFFER"."MODE SELECTION", in2 := 0)
   END_RUNG wire#w3
   // the same network as SCL:
   IF "AlwaysTRUE" THEN
       "RINSE-3_PUMP_CHASING"("SET TIME" := "SET_PARAMETERS"."RINSE-3_PUMP_CHASING_TIME_SV",   // "TIMING_BLOCK"
                              RESET := "RINSE-3_PUMP_CHASING".RESET,
                              INPUT := "AlwaysTRUE" AND ("BUFFER"."MODE SELECTION" = 1) AND ("BUFFER".PROCESS = 470) AND NOT "ERROR" AND NOT "CYCLE PAUSE",
                              "PRESENT VALUE OF TIME" => "SET_PARAMETERS"."RINSE-3_PUMP_CHASING_TIME_PV",
                              DONE => "RINSE-3_PUMP_CHASING".DONE);
   END_IF;
   "IEC_Timer_0_DB_31".TP(IN := ("BUFFER"."MODE SELECTION" = 1) AND ("BUFFER".PROCESS = 470) AND "RINSE-3_PUMP_CHASING".DONE,
                          PT := T#1S);
   IF "IEC_Timer_0_DB_31".Q THEN "BUFFER".PROCESS := 480; END_IF;
   IF ("BUFFER".PROCESS = 480) OR ("BUFFER"."MODE SELECTION" = 0) THEN
       "RINSE-3_PUMP_CHASING".DONE := FALSE;
   END_IF;
   "RINSE-3_PUMP_CHASING".RESET := ("BUFFER".PROCESS = 0) OR ("BUFFER"."MODE SELECTION" = 0);
END_REGION

REGION Network 50: NEXT CYCLE (FINAL_RINSE) POPUP
   RUNG wire#powerrail
      Contact( "AlwaysTRUE" )
      { S7_Templates := "SrcType := Int" } EQ_Contact(in1 := "BUFFER"."MODE SELECTION", in2 := 1)
      wire#w1
      { S7_Templates := "SrcType := Int" } EQ_Contact(in1 := "BUFFER".PROCESS, in2 := 480)
      wire#w2
      Contact( "RECIPE DB"."FINAL_RINSE-2_SELECT" )
      { S7_Templates := "time_type := Time" } "IEC_Timer_0_DB_11".TON(pt := T#5s, et =>)
      Move(in := 500, out1 => "BUFFER".PROCESS)
   END_RUNG
   RUNG wire#w2
      I_Contact( "RECIPE DB"."FINAL_RINSE-2_SELECT" )
      Move(in := 600, out1 => "BUFFER".PROCESS)
   END_RUNG
   RUNG wire#w1
      { S7_Templates := "SrcType := Int" } EQ_Contact(in1 := "BUFFER".PROCESS, in2 := 500)
      Contact( "CYCLE_POPUP".FINAL_RINSE_START_YES )
      Move(in := 510, out1 => "BUFFER".PROCESS)
   END_RUNG
   RUNG wire#w1
      { S7_Templates := "SrcType := Int" } EQ_Contact(in1 := "BUFFER".PROCESS, in2 := 500)
      Contact( "CYCLE_POPUP".FINAL_RINSE_START_NO )
      Move(in := 600, out1 => "BUFFER".PROCESS)
   END_RUNG
   // the same network as SCL:
   #_w1 := "AlwaysTRUE" AND ("BUFFER"."MODE SELECTION" = 1);
   #_w2 := #_w1 AND ("BUFFER".PROCESS = 480);
   "IEC_Timer_0_DB_11".TON(IN := #_w2 AND "RECIPE DB"."FINAL_RINSE-2_SELECT", PT := T#5s);
   IF "IEC_Timer_0_DB_11".Q THEN "BUFFER".PROCESS := 500; END_IF;
   IF #_w2 AND NOT "RECIPE DB"."FINAL_RINSE-2_SELECT" THEN "BUFFER".PROCESS := 600; END_IF;
   IF #_w1 AND ("BUFFER".PROCESS = 500) AND "CYCLE_POPUP".FINAL_RINSE_START_YES THEN
       "BUFFER".PROCESS := 510;
   END_IF;
   IF #_w1 AND ("BUFFER".PROCESS = 500) AND "CYCLE_POPUP".FINAL_RINSE_START_NO THEN
       "BUFFER".PROCESS := 600;
   END_IF;
END_REGION

REGION Network 51: PWT_LEVEL_CHECK
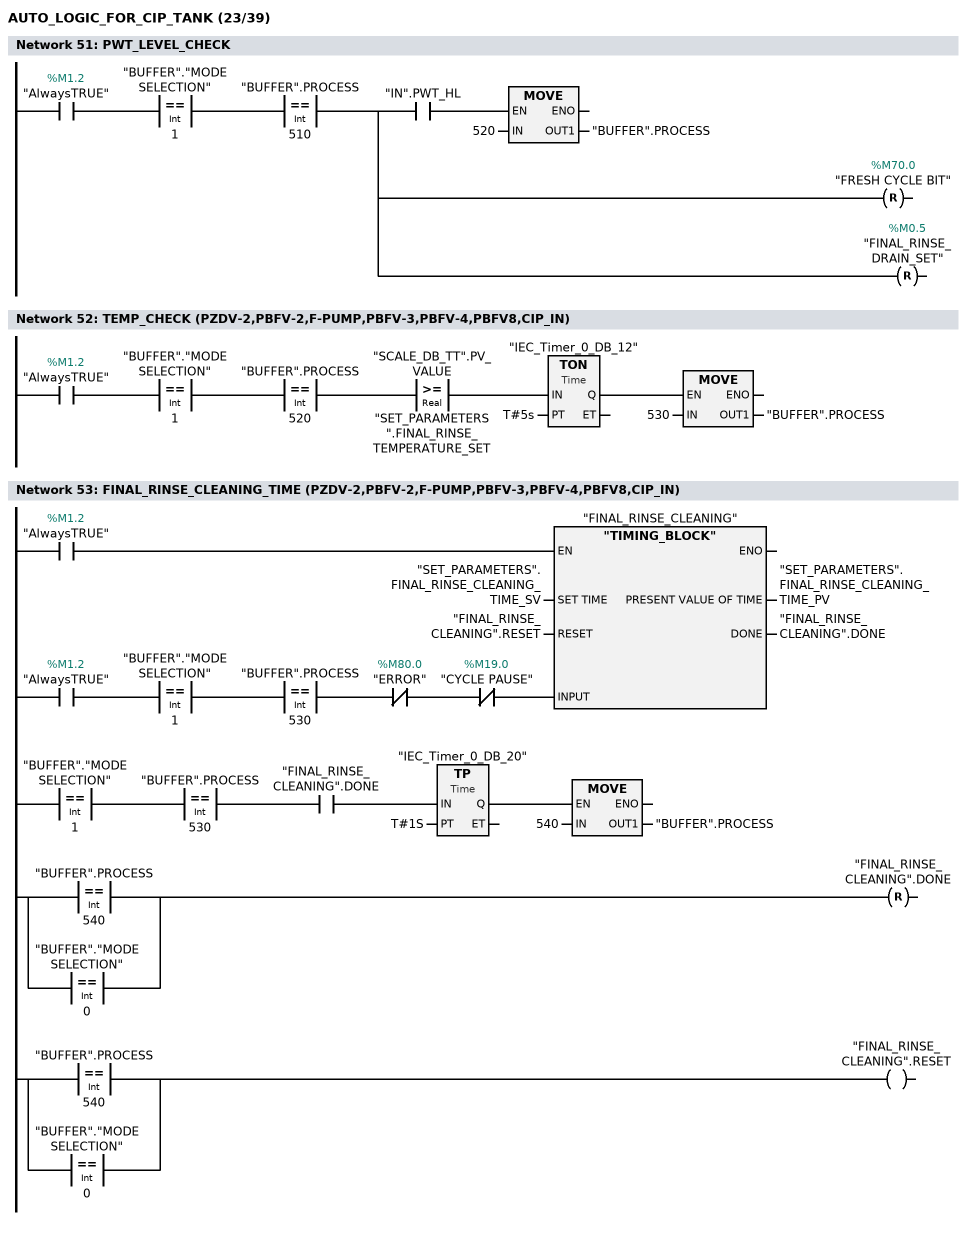
   RUNG wire#powerrail
      Contact( "AlwaysTRUE" )
      { S7_Templates := "SrcType := Int" } EQ_Contact(in1 := "BUFFER"."MODE SELECTION", in2 := 1)
      { S7_Templates := "SrcType := Int" } EQ_Contact(in1 := "BUFFER".PROCESS, in2 := 510)
      wire#w1
      Contact( "IN".PWT_HL )
      Move(in := 520, out1 => "BUFFER".PROCESS)
   END_RUNG
   RUNG wire#w1
      R_Coil( "FRESH CYCLE BIT" )
   END_RUNG
   RUNG wire#w1
      R_Coil( "FINAL_RINSE_DRAIN_SET" )
   END_RUNG
   // the same network as SCL:
   #_w1 := "AlwaysTRUE" AND ("BUFFER"."MODE SELECTION" = 1) AND ("BUFFER".PROCESS = 510);
   IF #_w1 AND "IN".PWT_HL THEN "BUFFER".PROCESS := 520; END_IF;
   IF #_w1 THEN
       "FRESH CYCLE BIT" := FALSE;
       "FINAL_RINSE_DRAIN_SET" := FALSE;
   END_IF;
END_REGION

REGION Network 52: TEMP_CHECK (PZDV-2,PBFV-2,F-PUMP,PBFV-3,PBFV-4,PBFV8,CIP_IN)
   RUNG wire#powerrail
      Contact( "AlwaysTRUE" )
      { S7_Templates := "SrcType := Int" } EQ_Contact(in1 := "BUFFER"."MODE SELECTION", in2 := 1)
      { S7_Templates := "SrcType := Int" } EQ_Contact(in1 := "BUFFER".PROCESS, in2 := 520)
      { S7_Templates := "SrcType := Real" } GE_Contact(in1 := "SCALE_DB_TT".PV_VALUE, in2 := "SET_PARAMETERS".FINAL_RINSE_TEMPERATURE_SET)
      { S7_Templates := "time_type := Time" } "IEC_Timer_0_DB_12".TON(pt := T#5s, et =>)
      Move(in := 530, out1 => "BUFFER".PROCESS)
   END_RUNG
   // the same network as SCL:
   "IEC_Timer_0_DB_12".TON(IN := "AlwaysTRUE" AND ("BUFFER"."MODE SELECTION" = 1) AND ("BUFFER".PROCESS = 520) AND ("SCALE_DB_TT".PV_VALUE >= "SET_PARAMETERS".FINAL_RINSE_TEMPERATURE_SET),
                           PT := T#5s);
   IF "IEC_Timer_0_DB_12".Q THEN "BUFFER".PROCESS := 530; END_IF;
END_REGION

REGION Network 53: FINAL_RINSE_CLEANING_TIME (PZDV-2,PBFV-2,F-PUMP,PBFV-3,PBFV-4,PBFV8,CIP_IN)
   RUNG wire#powerrail
      Contact( "AlwaysTRUE" )
      "FINAL_RINSE_CLEANING"(INPUT := wire#w1, "SET TIME" := "SET_PARAMETERS".FINAL_RINSE_CLEANING_TIME_SV, RESET := "FINAL_RINSE_CLEANING".RESET, "PRESENT VALUE OF TIME" => "SET_PARAMETERS".FINAL_RINSE_CLEANING_TIME_PV, DONE => "FINAL_RINSE_CLEANING".DONE)
   END_RUNG
   RUNG wire#powerrail
      Contact( "AlwaysTRUE" )
      { S7_Templates := "SrcType := Int" } EQ_Contact(in1 := "BUFFER"."MODE SELECTION", in2 := 1)
      { S7_Templates := "SrcType := Int" } EQ_Contact(in1 := "BUFFER".PROCESS, in2 := 530)
      I_Contact( "ERROR" )
      I_Contact( "CYCLE PAUSE" )
   END_RUNG wire#w1
   RUNG wire#powerrail
      { S7_Templates := "SrcType := Int" } EQ_Contact(in1 := "BUFFER"."MODE SELECTION", in2 := 1)
      { S7_Templates := "SrcType := Int" } EQ_Contact(in1 := "BUFFER".PROCESS, in2 := 530)
      Contact( "FINAL_RINSE_CLEANING".DONE )
      { S7_Templates := "time_type := Time" } "IEC_Timer_0_DB_20".TP(pt := T#1S, et =>)
      Move(in := 540, out1 => "BUFFER".PROCESS)
   END_RUNG
   RUNG wire#powerrail
      { S7_Templates := "SrcType := Int" } EQ_Contact(in1 := "BUFFER".PROCESS, in2 := 540)
      wire#w2
      R_Coil( "FINAL_RINSE_CLEANING".DONE )
   END_RUNG
   RUNG wire#powerrail
      { S7_Templates := "SrcType := Int" } EQ_Contact(in1 := "BUFFER"."MODE SELECTION", in2 := 0)
   END_RUNG wire#w2
   RUNG wire#powerrail
      { S7_Templates := "SrcType := Int" } EQ_Contact(in1 := "BUFFER".PROCESS, in2 := 540)
      wire#w3
      Coil( "FINAL_RINSE_CLEANING".RESET )
   END_RUNG
   RUNG wire#powerrail
      { S7_Templates := "SrcType := Int" } EQ_Contact(in1 := "BUFFER"."MODE SELECTION", in2 := 0)
   END_RUNG wire#w3
   // the same network as SCL:
   IF "AlwaysTRUE" THEN
       "FINAL_RINSE_CLEANING"("SET TIME" := "SET_PARAMETERS".FINAL_RINSE_CLEANING_TIME_SV,   // "TIMING_BLOCK"
                              RESET := "FINAL_RINSE_CLEANING".RESET,
                              INPUT := "AlwaysTRUE" AND ("BUFFER"."MODE SELECTION" = 1) AND ("BUFFER".PROCESS = 530) AND NOT "ERROR" AND NOT "CYCLE PAUSE",
                              "PRESENT VALUE OF TIME" => "SET_PARAMETERS".FINAL_RINSE_CLEANING_TIME_PV,
                              DONE => "FINAL_RINSE_CLEANING".DONE);
   END_IF;
   "IEC_Timer_0_DB_20".TP(IN := ("BUFFER"."MODE SELECTION" = 1) AND ("BUFFER".PROCESS = 530) AND "FINAL_RINSE_CLEANING".DONE,
                          PT := T#1S);
   IF "IEC_Timer_0_DB_20".Q THEN "BUFFER".PROCESS := 540; END_IF;
   IF ("BUFFER".PROCESS = 540) OR ("BUFFER"."MODE SELECTION" = 0) THEN
       "FINAL_RINSE_CLEANING".DONE := FALSE;
   END_IF;
   "FINAL_RINSE_CLEANING".RESET := ("BUFFER".PROCESS = 540) OR ("BUFFER"."MODE SELECTION" = 0);
END_REGION

REGION Network 54: CONDUCTIVITY ACHIEVED OR NOT ACHIEVED BIT SET
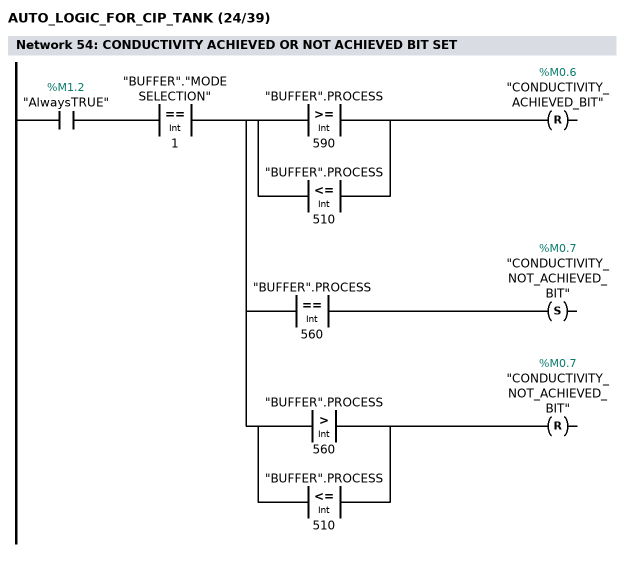
   RUNG wire#powerrail
      Contact( "AlwaysTRUE" )
      { S7_Templates := "SrcType := Int" } EQ_Contact(in1 := "BUFFER"."MODE SELECTION", in2 := 1)
      wire#w1
      { S7_Templates := "SrcType := Int" } GE_Contact(in1 := "BUFFER".PROCESS, in2 := 590)
      wire#w2
      R_Coil( "CONDUCTIVITY_ACHIEVED_BIT" )
   END_RUNG
   RUNG wire#w1
      { S7_Templates := "SrcType := Int" } LE_Contact(in1 := "BUFFER".PROCESS, in2 := 510)
   END_RUNG wire#w2
   RUNG wire#w1
      { S7_Templates := "SrcType := Int" } EQ_Contact(in1 := "BUFFER".PROCESS, in2 := 560)
      S_Coil( "CONDUCTIVITY_NOT_ACHIEVED_BIT" )
   END_RUNG
   RUNG wire#w1
      { S7_Templates := "SrcType := Int" } GT_Contact(in1 := "BUFFER".PROCESS, in2 := 560)
      wire#w3
      R_Coil( "CONDUCTIVITY_NOT_ACHIEVED_BIT" )
   END_RUNG
   RUNG wire#w1
      { S7_Templates := "SrcType := Int" } LE_Contact(in1 := "BUFFER".PROCESS, in2 := 510)
   END_RUNG wire#w3
   // the same network as SCL:
   #_w1 := "AlwaysTRUE" AND ("BUFFER"."MODE SELECTION" = 1);
   IF #_w1 AND (("BUFFER".PROCESS >= 590) OR ("BUFFER".PROCESS <= 510)) THEN
       "CONDUCTIVITY_ACHIEVED_BIT" := FALSE;
   END_IF;
   IF #_w1 AND ("BUFFER".PROCESS = 560) THEN "CONDUCTIVITY_NOT_ACHIEVED_BIT" := TRUE; END_IF;
   IF #_w1 AND (("BUFFER".PROCESS > 560) OR ("BUFFER".PROCESS <= 510)) THEN
       "CONDUCTIVITY_NOT_ACHIEVED_BIT" := FALSE;
   END_IF;
END_REGION

REGION Network 55: FINAL_RINSE_CONDUCTIVITY CHECKING TIME
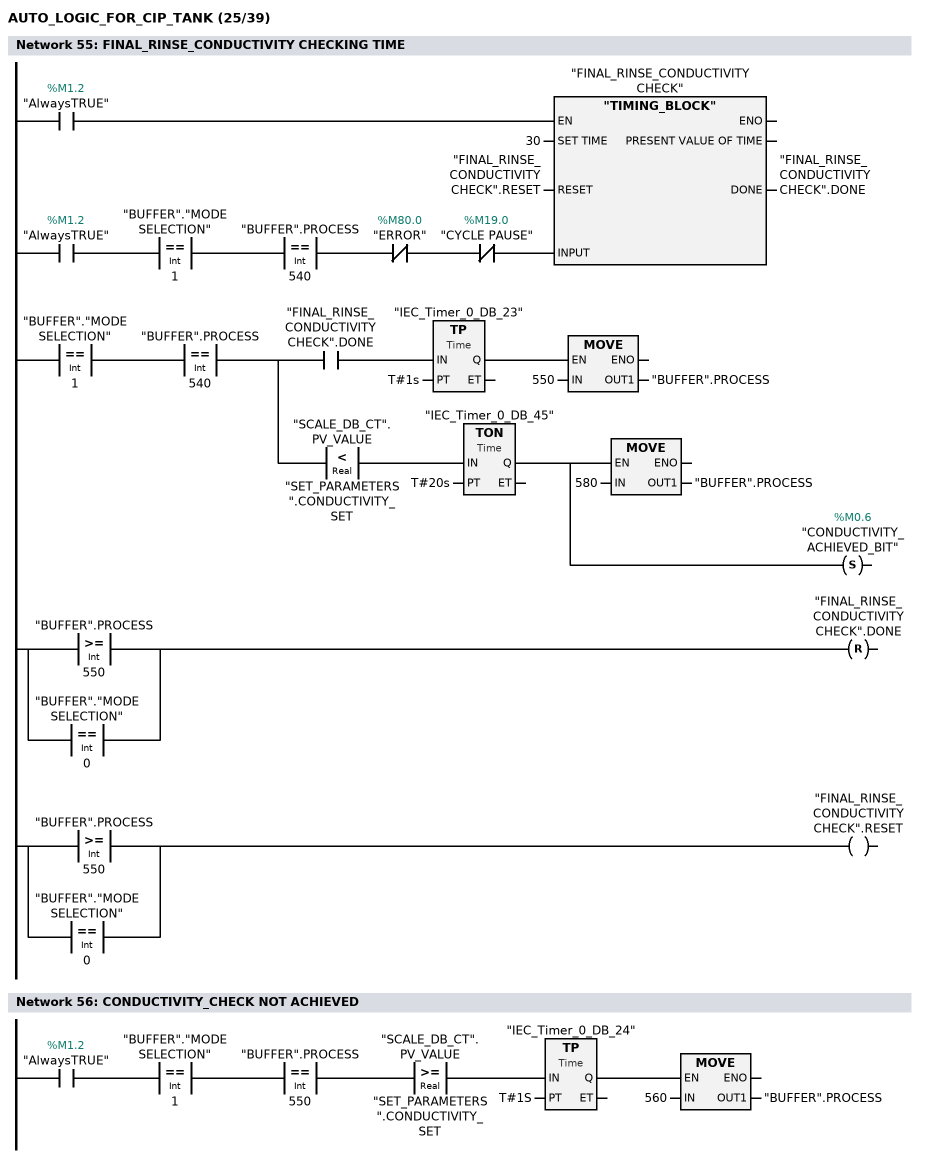
   RUNG wire#powerrail
      Contact( "AlwaysTRUE" )
      "FINAL_RINSE_CONDUCTIVITY CHECK"(INPUT := wire#w1, "SET TIME" := 30, RESET := "FINAL_RINSE_CONDUCTIVITY CHECK".RESET, "PRESENT VALUE OF TIME" =>, DONE => "FINAL_RINSE_CONDUCTIVITY CHECK".DONE)
   END_RUNG
   RUNG wire#powerrail
      Contact( "AlwaysTRUE" )
      { S7_Templates := "SrcType := Int" } EQ_Contact(in1 := "BUFFER"."MODE SELECTION", in2 := 1)
      { S7_Templates := "SrcType := Int" } EQ_Contact(in1 := "BUFFER".PROCESS, in2 := 540)
      I_Contact( "ERROR" )
      I_Contact( "CYCLE PAUSE" )
   END_RUNG wire#w1
   RUNG wire#powerrail
      { S7_Templates := "SrcType := Int" } EQ_Contact(in1 := "BUFFER"."MODE SELECTION", in2 := 1)
      { S7_Templates := "SrcType := Int" } EQ_Contact(in1 := "BUFFER".PROCESS, in2 := 540)
      wire#w2
      Contact( "FINAL_RINSE_CONDUCTIVITY CHECK".DONE )
      { S7_Templates := "time_type := Time" } "IEC_Timer_0_DB_23".TP(pt := T#1s, et =>)
      Move(in := 550, out1 => "BUFFER".PROCESS)
   END_RUNG
   RUNG wire#w2
      { S7_Templates := "SrcType := Real" } LT_Contact(in1 := "SCALE_DB_CT".PV_VALUE, in2 := "SET_PARAMETERS".CONDUCTIVITY_SET)
      { S7_Templates := "time_type := Time" } "IEC_Timer_0_DB_45".TON(pt := T#20s, et =>)
      wire#w3
      Move(in := 580, out1 => "BUFFER".PROCESS)
   END_RUNG
   RUNG wire#w3
      S_Coil( "CONDUCTIVITY_ACHIEVED_BIT" )
   END_RUNG
   RUNG wire#powerrail
      { S7_Templates := "SrcType := Int" } GE_Contact(in1 := "BUFFER".PROCESS, in2 := 550)
      wire#w4
      R_Coil( "FINAL_RINSE_CONDUCTIVITY CHECK".DONE )
   END_RUNG
   RUNG wire#powerrail
      { S7_Templates := "SrcType := Int" } EQ_Contact(in1 := "BUFFER"."MODE SELECTION", in2 := 0)
   END_RUNG wire#w4
   RUNG wire#powerrail
      { S7_Templates := "SrcType := Int" } GE_Contact(in1 := "BUFFER".PROCESS, in2 := 550)
      wire#w5
      Coil( "FINAL_RINSE_CONDUCTIVITY CHECK".RESET )
   END_RUNG
   RUNG wire#powerrail
      { S7_Templates := "SrcType := Int" } EQ_Contact(in1 := "BUFFER"."MODE SELECTION", in2 := 0)
   END_RUNG wire#w5
   // the same network as SCL:
   IF "AlwaysTRUE" THEN
       "FINAL_RINSE_CONDUCTIVITY CHECK"("SET TIME" := 30,   // "TIMING_BLOCK"
                               RESET := "FINAL_RINSE_CONDUCTIVITY CHECK".RESET,
                               INPUT := "AlwaysTRUE" AND ("BUFFER"."MODE SELECTION" = 1) AND ("BUFFER".PROCESS = 540) AND NOT "ERROR" AND NOT "CYCLE PAUSE",
                               DONE => "FINAL_RINSE_CONDUCTIVITY CHECK".DONE);
   END_IF;
   #_w1 := ("BUFFER"."MODE SELECTION" = 1) AND ("BUFFER".PROCESS = 540);
   "IEC_Timer_0_DB_23".TP(IN := #_w1 AND "FINAL_RINSE_CONDUCTIVITY CHECK".DONE, PT := T#1s);
   IF "IEC_Timer_0_DB_23".Q THEN "BUFFER".PROCESS := 550; END_IF;
   "IEC_Timer_0_DB_45".TON(IN := #_w1 AND ("SCALE_DB_CT".PV_VALUE < "SET_PARAMETERS".CONDUCTIVITY_SET),
                           PT := T#20s);
   IF "IEC_Timer_0_DB_45".Q THEN
       "BUFFER".PROCESS := 580;
       "CONDUCTIVITY_ACHIEVED_BIT" := TRUE;
   END_IF;
   IF ("BUFFER".PROCESS >= 550) OR ("BUFFER"."MODE SELECTION" = 0) THEN
       "FINAL_RINSE_CONDUCTIVITY CHECK".DONE := FALSE;
   END_IF;
   "FINAL_RINSE_CONDUCTIVITY CHECK".RESET := ("BUFFER".PROCESS >= 550) OR ("BUFFER"."MODE SELECTION" = 0);
END_REGION

REGION Network 56: CONDUCTIVITY_CHECK NOT ACHIEVED
   RUNG wire#powerrail
      Contact( "AlwaysTRUE" )
      { S7_Templates := "SrcType := Int" } EQ_Contact(in1 := "BUFFER"."MODE SELECTION", in2 := 1)
      { S7_Templates := "SrcType := Int" } EQ_Contact(in1 := "BUFFER".PROCESS, in2 := 550)
      { S7_Templates := "SrcType := Real" } GE_Contact(in1 := "SCALE_DB_CT".PV_VALUE, in2 := "SET_PARAMETERS".CONDUCTIVITY_SET)
      { S7_Templates := "time_type := Time" } "IEC_Timer_0_DB_24".TP(pt := T#1S, et =>)
      Move(in := 560, out1 => "BUFFER".PROCESS)
   END_RUNG
   // the same network as SCL:
   "IEC_Timer_0_DB_24".TP(IN := "AlwaysTRUE" AND ("BUFFER"."MODE SELECTION" = 1) AND ("BUFFER".PROCESS = 550) AND ("SCALE_DB_CT".PV_VALUE >= "SET_PARAMETERS".CONDUCTIVITY_SET),
                          PT := T#1S);
   IF "IEC_Timer_0_DB_24".Q THEN "BUFFER".PROCESS := 560; END_IF;
END_REGION

REGION Network 57: RECIRCULATION_OR_FRESH CYCLE_ OR DRAIN POPUP
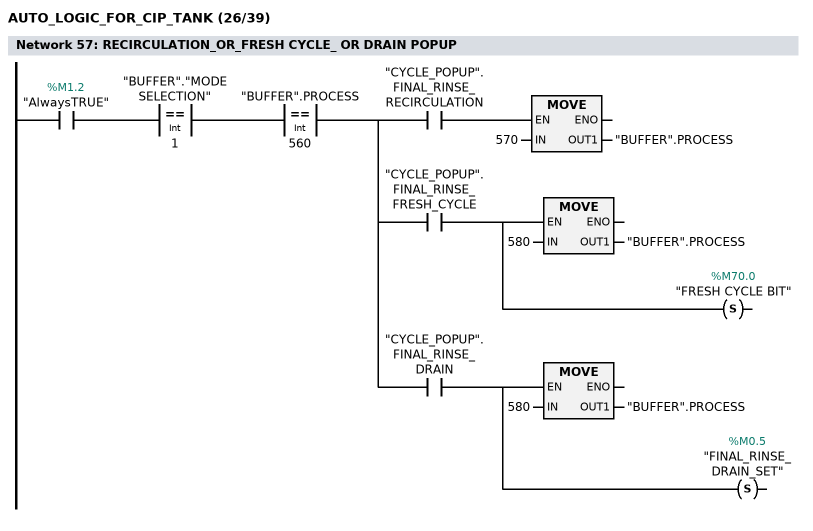
   RUNG wire#powerrail
      Contact( "AlwaysTRUE" )
      { S7_Templates := "SrcType := Int" } EQ_Contact(in1 := "BUFFER"."MODE SELECTION", in2 := 1)
      { S7_Templates := "SrcType := Int" } EQ_Contact(in1 := "BUFFER".PROCESS, in2 := 560)
      wire#w1
      Contact( "CYCLE_POPUP".FINAL_RINSE_RECIRCULATION )
      Move(in := 570, out1 => "BUFFER".PROCESS)
   END_RUNG
   RUNG wire#w1
      Contact( "CYCLE_POPUP".FINAL_RINSE_FRESH_CYCLE )
      wire#w2
      Move(in := 580, out1 => "BUFFER".PROCESS)
   END_RUNG
   RUNG wire#w2
      S_Coil( "FRESH CYCLE BIT" )
   END_RUNG
   RUNG wire#w1
      Contact( "CYCLE_POPUP".FINAL_RINSE_DRAIN )
      wire#w3
      Move(in := 580, out1 => "BUFFER".PROCESS)
   END_RUNG
   RUNG wire#w3
      S_Coil( "FINAL_RINSE_DRAIN_SET" )
   END_RUNG
   // the same network as SCL:
   #_w1 := "AlwaysTRUE" AND ("BUFFER"."MODE SELECTION" = 1) AND ("BUFFER".PROCESS = 560);
   IF #_w1 AND "CYCLE_POPUP".FINAL_RINSE_RECIRCULATION THEN "BUFFER".PROCESS := 570; END_IF;
   IF #_w1 AND "CYCLE_POPUP".FINAL_RINSE_FRESH_CYCLE THEN
       "BUFFER".PROCESS := 580;
       "FRESH CYCLE BIT" := TRUE;
   END_IF;
   IF #_w1 AND "CYCLE_POPUP".FINAL_RINSE_DRAIN THEN
       "BUFFER".PROCESS := 580;
       "FINAL_RINSE_DRAIN_SET" := TRUE;
   END_IF;
END_REGION

REGION Network 58: FINAL_RINSE_RECIRCULATION_TIME (CIP-OUT,R-PUMP,PBFV-6,PBFV-8,CIP-IN)
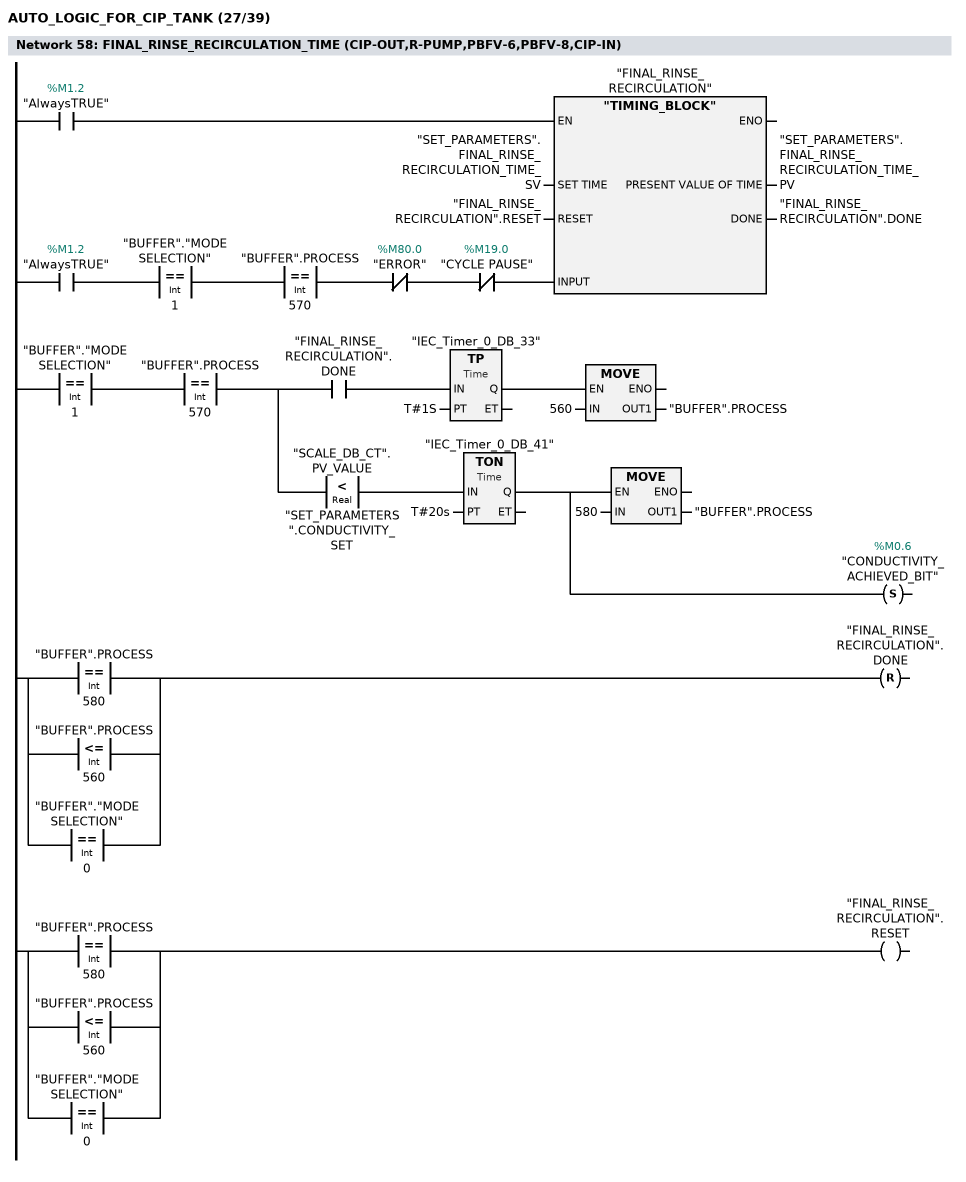
   RUNG wire#powerrail
      Contact( "AlwaysTRUE" )
      "FINAL_RINSE_RECIRCULATION"(INPUT := wire#w1, "SET TIME" := "SET_PARAMETERS".FINAL_RINSE_RECIRCULATION_TIME_SV, RESET := "FINAL_RINSE_RECIRCULATION".RESET, "PRESENT VALUE OF TIME" => "SET_PARAMETERS".FINAL_RINSE_RECIRCULATION_TIME_PV, DONE => "FINAL_RINSE_RECIRCULATION".DONE)
   END_RUNG
   RUNG wire#powerrail
      Contact( "AlwaysTRUE" )
      { S7_Templates := "SrcType := Int" } EQ_Contact(in1 := "BUFFER"."MODE SELECTION", in2 := 1)
      { S7_Templates := "SrcType := Int" } EQ_Contact(in1 := "BUFFER".PROCESS, in2 := 570)
      I_Contact( "ERROR" )
      I_Contact( "CYCLE PAUSE" )
   END_RUNG wire#w1
   RUNG wire#powerrail
      { S7_Templates := "SrcType := Int" } EQ_Contact(in1 := "BUFFER"."MODE SELECTION", in2 := 1)
      { S7_Templates := "SrcType := Int" } EQ_Contact(in1 := "BUFFER".PROCESS, in2 := 570)
      wire#w2
      Contact( "FINAL_RINSE_RECIRCULATION".DONE )
      { S7_Templates := "time_type := Time" } "IEC_Timer_0_DB_33".TP(pt := T#1S, et =>)
      Move(in := 560, out1 => "BUFFER".PROCESS)
   END_RUNG
   RUNG wire#w2
      { S7_Templates := "SrcType := Real" } LT_Contact(in1 := "SCALE_DB_CT".PV_VALUE, in2 := "SET_PARAMETERS".CONDUCTIVITY_SET)
      { S7_Templates := "time_type := Time" } "IEC_Timer_0_DB_41".TON(pt := T#20s, et =>)
      wire#w3
      Move(in := 580, out1 => "BUFFER".PROCESS)
   END_RUNG
   RUNG wire#w3
      S_Coil( "CONDUCTIVITY_ACHIEVED_BIT" )
   END_RUNG
   RUNG wire#powerrail
      { S7_Templates := "SrcType := Int" } EQ_Contact(in1 := "BUFFER".PROCESS, in2 := 580)
      wire#w4
      R_Coil( "FINAL_RINSE_RECIRCULATION".DONE )
   END_RUNG
   RUNG wire#powerrail
      { S7_Templates := "SrcType := Int" } LE_Contact(in1 := "BUFFER".PROCESS, in2 := 560)
   END_RUNG wire#w4
   RUNG wire#powerrail
      { S7_Templates := "SrcType := Int" } EQ_Contact(in1 := "BUFFER"."MODE SELECTION", in2 := 0)
   END_RUNG wire#w4
   RUNG wire#powerrail
      { S7_Templates := "SrcType := Int" } EQ_Contact(in1 := "BUFFER".PROCESS, in2 := 580)
      wire#w5
      Coil( "FINAL_RINSE_RECIRCULATION".RESET )
   END_RUNG
   RUNG wire#powerrail
      { S7_Templates := "SrcType := Int" } LE_Contact(in1 := "BUFFER".PROCESS, in2 := 560)
   END_RUNG wire#w5
   RUNG wire#powerrail
      { S7_Templates := "SrcType := Int" } EQ_Contact(in1 := "BUFFER"."MODE SELECTION", in2 := 0)
   END_RUNG wire#w5
   // the same network as SCL:
   IF "AlwaysTRUE" THEN
       "FINAL_RINSE_RECIRCULATION"("SET TIME" := "SET_PARAMETERS".FINAL_RINSE_RECIRCULATION_TIME_SV,   // "TIMING_BLOCK"
                               RESET := "FINAL_RINSE_RECIRCULATION".RESET,
                               INPUT := "AlwaysTRUE" AND ("BUFFER"."MODE SELECTION" = 1) AND ("BUFFER".PROCESS = 570) AND NOT "ERROR" AND NOT "CYCLE PAUSE",
                               "PRESENT VALUE OF TIME" => "SET_PARAMETERS".FINAL_RINSE_RECIRCULATION_TIME_PV,
                               DONE => "FINAL_RINSE_RECIRCULATION".DONE);
   END_IF;
   #_w1 := ("BUFFER"."MODE SELECTION" = 1) AND ("BUFFER".PROCESS = 570);
   "IEC_Timer_0_DB_33".TP(IN := #_w1 AND "FINAL_RINSE_RECIRCULATION".DONE, PT := T#1S);
   IF "IEC_Timer_0_DB_33".Q THEN "BUFFER".PROCESS := 560; END_IF;
   "IEC_Timer_0_DB_41".TON(IN := #_w1 AND ("SCALE_DB_CT".PV_VALUE < "SET_PARAMETERS".CONDUCTIVITY_SET),
                           PT := T#20s);
   IF "IEC_Timer_0_DB_41".Q THEN
       "BUFFER".PROCESS := 580;
       "CONDUCTIVITY_ACHIEVED_BIT" := TRUE;
   END_IF;
   IF ("BUFFER".PROCESS = 580) OR ("BUFFER".PROCESS <= 560) OR ("BUFFER"."MODE SELECTION" = 0) THEN
       "FINAL_RINSE_RECIRCULATION".DONE := FALSE;
   END_IF;
   "FINAL_RINSE_RECIRCULATION".RESET := ("BUFFER".PROCESS = 580) OR ("BUFFER".PROCESS <= 560) OR ("BUFFER"."MODE SELECTION" = 0);
END_REGION

REGION Network 59: FINAL_RINSE_DRAIN_TIME (CIP-OUT,R_PUMP,PBFV-11)
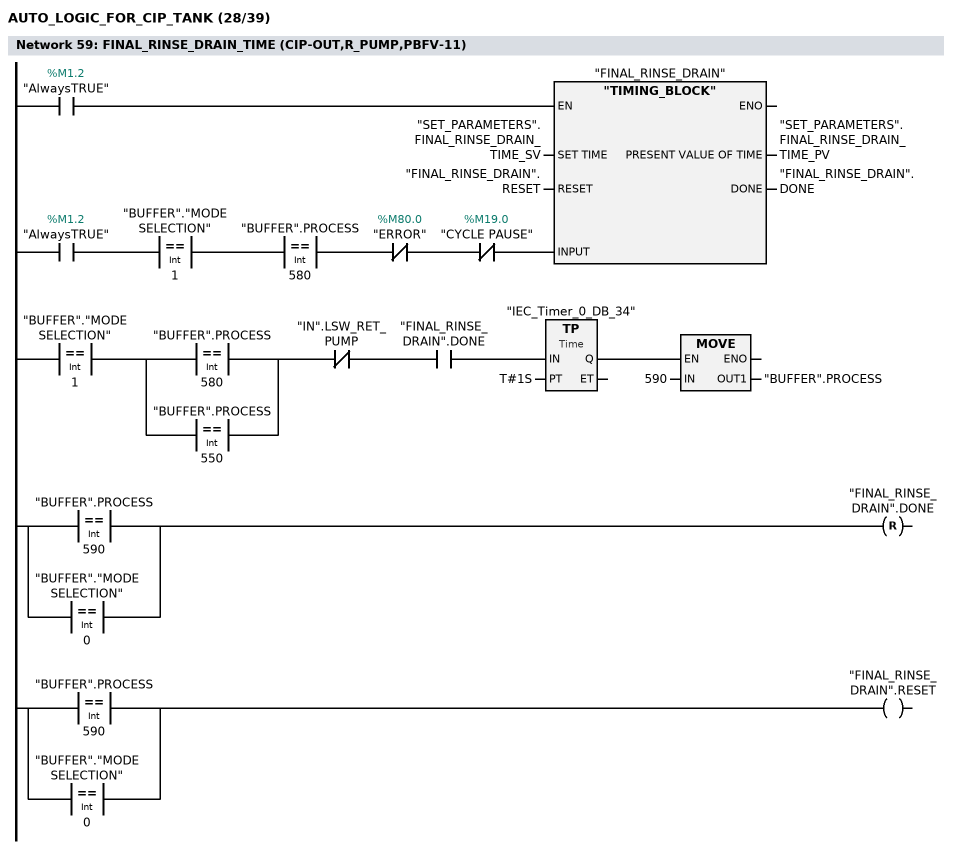
   RUNG wire#powerrail
      Contact( "AlwaysTRUE" )
      "FINAL_RINSE_DRAIN"(INPUT := wire#w1, "SET TIME" := "SET_PARAMETERS".FINAL_RINSE_DRAIN_TIME_SV, RESET := "FINAL_RINSE_DRAIN".RESET, "PRESENT VALUE OF TIME" => "SET_PARAMETERS".FINAL_RINSE_DRAIN_TIME_PV, DONE => "FINAL_RINSE_DRAIN".DONE)
   END_RUNG
   RUNG wire#powerrail
      Contact( "AlwaysTRUE" )
      { S7_Templates := "SrcType := Int" } EQ_Contact(in1 := "BUFFER"."MODE SELECTION", in2 := 1)
      { S7_Templates := "SrcType := Int" } EQ_Contact(in1 := "BUFFER".PROCESS, in2 := 580)
      I_Contact( "ERROR" )
      I_Contact( "CYCLE PAUSE" )
   END_RUNG wire#w1
   RUNG wire#powerrail
      { S7_Templates := "SrcType := Int" } EQ_Contact(in1 := "BUFFER"."MODE SELECTION", in2 := 1)
      wire#w2
      { S7_Templates := "SrcType := Int" } EQ_Contact(in1 := "BUFFER".PROCESS, in2 := 580)
      wire#w3
      I_Contact( "IN".LSW_RET_PUMP )
      Contact( "FINAL_RINSE_DRAIN".DONE )
      { S7_Templates := "time_type := Time" } "IEC_Timer_0_DB_34".TP(pt := T#1S, et =>)
      Move(in := 590, out1 => "BUFFER".PROCESS)
   END_RUNG
   RUNG wire#w2
      { S7_Templates := "SrcType := Int" } EQ_Contact(in1 := "BUFFER".PROCESS, in2 := 550)
   END_RUNG wire#w3
   RUNG wire#powerrail
      { S7_Templates := "SrcType := Int" } EQ_Contact(in1 := "BUFFER".PROCESS, in2 := 590)
      wire#w4
      R_Coil( "FINAL_RINSE_DRAIN".DONE )
   END_RUNG
   RUNG wire#powerrail
      { S7_Templates := "SrcType := Int" } EQ_Contact(in1 := "BUFFER"."MODE SELECTION", in2 := 0)
   END_RUNG wire#w4
   RUNG wire#powerrail
      { S7_Templates := "SrcType := Int" } EQ_Contact(in1 := "BUFFER".PROCESS, in2 := 590)
      wire#w5
      Coil( "FINAL_RINSE_DRAIN".RESET )
   END_RUNG
   RUNG wire#powerrail
      { S7_Templates := "SrcType := Int" } EQ_Contact(in1 := "BUFFER"."MODE SELECTION", in2 := 0)
   END_RUNG wire#w5
   // the same network as SCL:
   IF "AlwaysTRUE" THEN
       "FINAL_RINSE_DRAIN"("SET TIME" := "SET_PARAMETERS".FINAL_RINSE_DRAIN_TIME_SV,   // "TIMING_BLOCK"
                           RESET := "FINAL_RINSE_DRAIN".RESET,
                           INPUT := "AlwaysTRUE" AND ("BUFFER"."MODE SELECTION" = 1) AND ("BUFFER".PROCESS = 580) AND NOT "ERROR" AND NOT "CYCLE PAUSE",
                           "PRESENT VALUE OF TIME" => "SET_PARAMETERS".FINAL_RINSE_DRAIN_TIME_PV,
                           DONE => "FINAL_RINSE_DRAIN".DONE);
   END_IF;
   "IEC_Timer_0_DB_34".TP(IN := ("BUFFER"."MODE SELECTION" = 1) AND (("BUFFER".PROCESS = 580) OR ("BUFFER".PROCESS = 550)) AND NOT "IN".LSW_RET_PUMP AND "FINAL_RINSE_DRAIN".DONE,
                          PT := T#1S);
   IF "IEC_Timer_0_DB_34".Q THEN "BUFFER".PROCESS := 590; END_IF;
   IF ("BUFFER".PROCESS = 590) OR ("BUFFER"."MODE SELECTION" = 0) THEN
       "FINAL_RINSE_DRAIN".DONE := FALSE;
   END_IF;
   "FINAL_RINSE_DRAIN".RESET := ("BUFFER".PROCESS = 590) OR ("BUFFER"."MODE SELECTION" = 0);
END_REGION

REGION Network 60: FINAL_RINSE_PUMP_CHASING_TIME (PBFV-12,PBFV13)
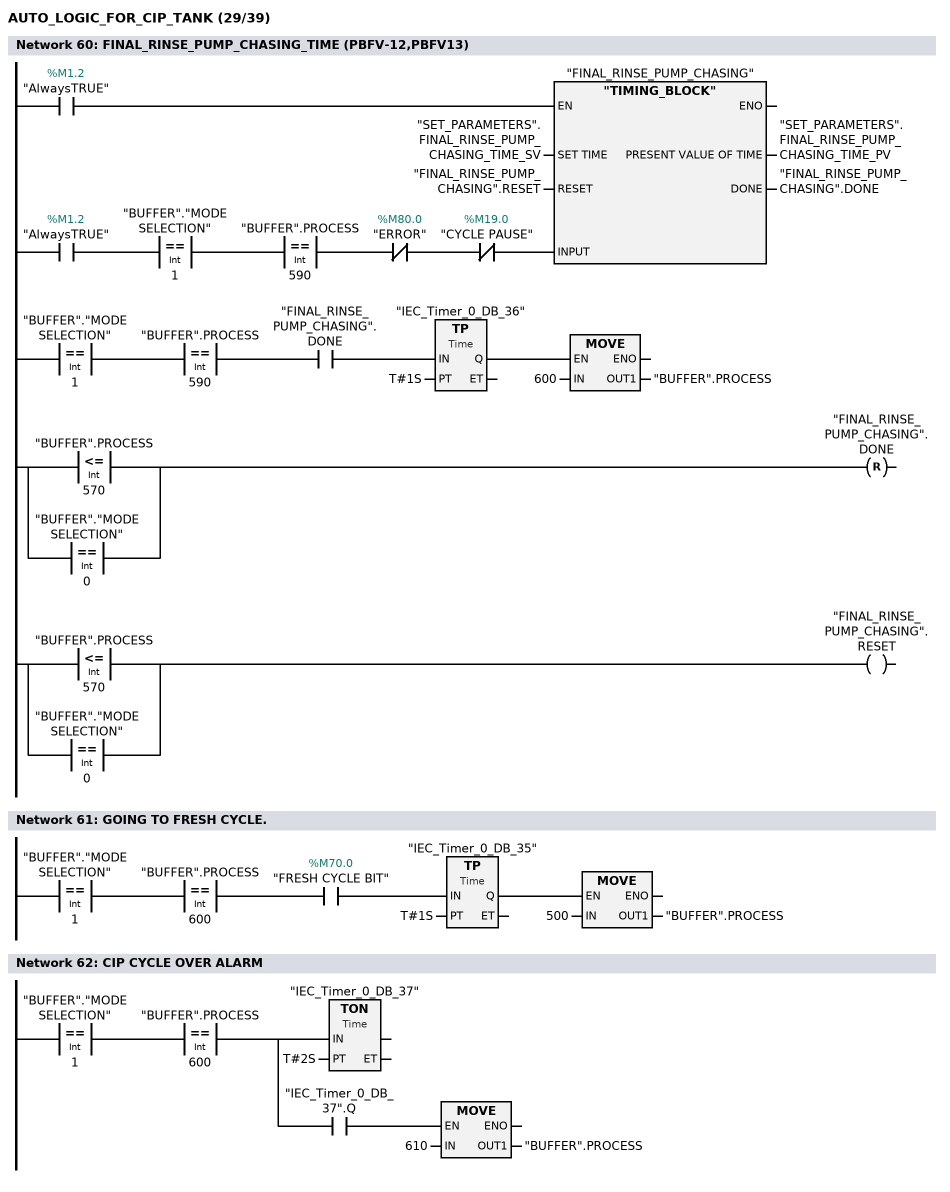
   RUNG wire#powerrail
      Contact( "AlwaysTRUE" )
      "FINAL_RINSE_PUMP_CHASING"(INPUT := wire#w1, "SET TIME" := "SET_PARAMETERS".FINAL_RINSE_PUMP_CHASING_TIME_SV, RESET := "FINAL_RINSE_PUMP_CHASING".RESET, "PRESENT VALUE OF TIME" => "SET_PARAMETERS".FINAL_RINSE_PUMP_CHASING_TIME_PV, DONE => "FINAL_RINSE_PUMP_CHASING".DONE)
   END_RUNG
   RUNG wire#powerrail
      Contact( "AlwaysTRUE" )
      { S7_Templates := "SrcType := Int" } EQ_Contact(in1 := "BUFFER"."MODE SELECTION", in2 := 1)
      { S7_Templates := "SrcType := Int" } EQ_Contact(in1 := "BUFFER".PROCESS, in2 := 590)
      I_Contact( "ERROR" )
      I_Contact( "CYCLE PAUSE" )
   END_RUNG wire#w1
   RUNG wire#powerrail
      { S7_Templates := "SrcType := Int" } EQ_Contact(in1 := "BUFFER"."MODE SELECTION", in2 := 1)
      { S7_Templates := "SrcType := Int" } EQ_Contact(in1 := "BUFFER".PROCESS, in2 := 590)
      Contact( "FINAL_RINSE_PUMP_CHASING".DONE )
      { S7_Templates := "time_type := Time" } "IEC_Timer_0_DB_36".TP(pt := T#1S, et =>)
      Move(in := 600, out1 => "BUFFER".PROCESS)
   END_RUNG
   RUNG wire#powerrail
      { S7_Templates := "SrcType := Int" } LE_Contact(in1 := "BUFFER".PROCESS, in2 := 570)
      wire#w2
      R_Coil( "FINAL_RINSE_PUMP_CHASING".DONE )
   END_RUNG
   RUNG wire#powerrail
      { S7_Templates := "SrcType := Int" } EQ_Contact(in1 := "BUFFER"."MODE SELECTION", in2 := 0)
   END_RUNG wire#w2
   RUNG wire#powerrail
      { S7_Templates := "SrcType := Int" } LE_Contact(in1 := "BUFFER".PROCESS, in2 := 570)
      wire#w3
      Coil( "FINAL_RINSE_PUMP_CHASING".RESET )
   END_RUNG
   RUNG wire#powerrail
      { S7_Templates := "SrcType := Int" } EQ_Contact(in1 := "BUFFER"."MODE SELECTION", in2 := 0)
   END_RUNG wire#w3
   // the same network as SCL:
   IF "AlwaysTRUE" THEN
       "FINAL_RINSE_PUMP_CHASING"("SET TIME" := "SET_PARAMETERS".FINAL_RINSE_PUMP_CHASING_TIME_SV,   // "TIMING_BLOCK"
                               RESET := "FINAL_RINSE_PUMP_CHASING".RESET,
                               INPUT := "AlwaysTRUE" AND ("BUFFER"."MODE SELECTION" = 1) AND ("BUFFER".PROCESS = 590) AND NOT "ERROR" AND NOT "CYCLE PAUSE",
                               "PRESENT VALUE OF TIME" => "SET_PARAMETERS".FINAL_RINSE_PUMP_CHASING_TIME_PV,
                               DONE => "FINAL_RINSE_PUMP_CHASING".DONE);
   END_IF;
   "IEC_Timer_0_DB_36".TP(IN := ("BUFFER"."MODE SELECTION" = 1) AND ("BUFFER".PROCESS = 590) AND "FINAL_RINSE_PUMP_CHASING".DONE,
                          PT := T#1S);
   IF "IEC_Timer_0_DB_36".Q THEN "BUFFER".PROCESS := 600; END_IF;
   IF ("BUFFER".PROCESS <= 570) OR ("BUFFER"."MODE SELECTION" = 0) THEN
       "FINAL_RINSE_PUMP_CHASING".DONE := FALSE;
   END_IF;
   "FINAL_RINSE_PUMP_CHASING".RESET := ("BUFFER".PROCESS <= 570) OR ("BUFFER"."MODE SELECTION" = 0);
END_REGION

REGION Network 61: GOING TO FRESH CYCLE.
   RUNG wire#powerrail
      { S7_Templates := "SrcType := Int" } EQ_Contact(in1 := "BUFFER"."MODE SELECTION", in2 := 1)
      { S7_Templates := "SrcType := Int" } EQ_Contact(in1 := "BUFFER".PROCESS, in2 := 600)
      Contact( "FRESH CYCLE BIT" )
      { S7_Templates := "time_type := Time" } "IEC_Timer_0_DB_35".TP(pt := T#1S, et =>)
      Move(in := 500, out1 => "BUFFER".PROCESS)
   END_RUNG
   // the same network as SCL:
   "IEC_Timer_0_DB_35".TP(IN := ("BUFFER"."MODE SELECTION" = 1) AND ("BUFFER".PROCESS = 600) AND "FRESH CYCLE BIT",
                          PT := T#1S);
   IF "IEC_Timer_0_DB_35".Q THEN "BUFFER".PROCESS := 500; END_IF;
END_REGION

REGION Network 62: CIP CYCLE OVER ALARM
   RUNG wire#powerrail
      { S7_Templates := "SrcType := Int" } EQ_Contact(in1 := "BUFFER"."MODE SELECTION", in2 := 1)
      { S7_Templates := "SrcType := Int" } EQ_Contact(in1 := "BUFFER".PROCESS, in2 := 600)
      wire#w1
      { S7_Templates := "time_type := Time" } "IEC_Timer_0_DB_37".TON(pt := T#2S, et =>)
   END_RUNG
   RUNG wire#w1
      Contact( "IEC_Timer_0_DB_37".Q )
      Move(in := 610, out1 => "BUFFER".PROCESS)
   END_RUNG
   // the same network as SCL:
   #_w1 := ("BUFFER"."MODE SELECTION" = 1) AND ("BUFFER".PROCESS = 600);
   "IEC_Timer_0_DB_37".TON(IN := #_w1, PT := T#2S);
   IF #_w1 AND "IEC_Timer_0_DB_37".Q THEN "BUFFER".PROCESS := 610; END_IF;
END_REGION

REGION Network 63: CIP CYCLE OVER
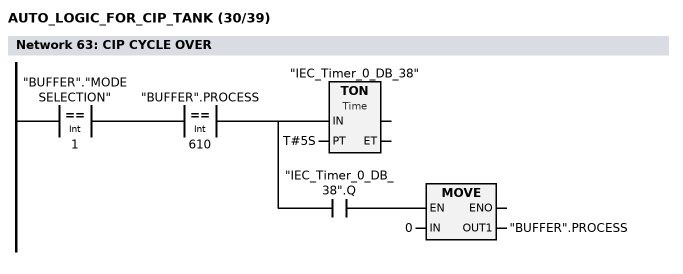
   RUNG wire#powerrail
      { S7_Templates := "SrcType := Int" } EQ_Contact(in1 := "BUFFER"."MODE SELECTION", in2 := 1)
      { S7_Templates := "SrcType := Int" } EQ_Contact(in1 := "BUFFER".PROCESS, in2 := 610)
      wire#w1
      { S7_Templates := "time_type := Time" } "IEC_Timer_0_DB_38".TON(pt := T#5S, et =>)
   END_RUNG
   RUNG wire#w1
      Contact( "IEC_Timer_0_DB_38".Q )
      Move(in := 0, out1 => "BUFFER".PROCESS)
   END_RUNG
   // the same network as SCL:
   #_w1 := ("BUFFER"."MODE SELECTION" = 1) AND ("BUFFER".PROCESS = 610);
   "IEC_Timer_0_DB_38".TON(IN := #_w1, PT := T#5S);
   IF #_w1 AND "IEC_Timer_0_DB_38".Q THEN "BUFFER".PROCESS := 0; END_IF;
END_REGION

REGION Network 65: CONDANSATE VALVE ON TIMER
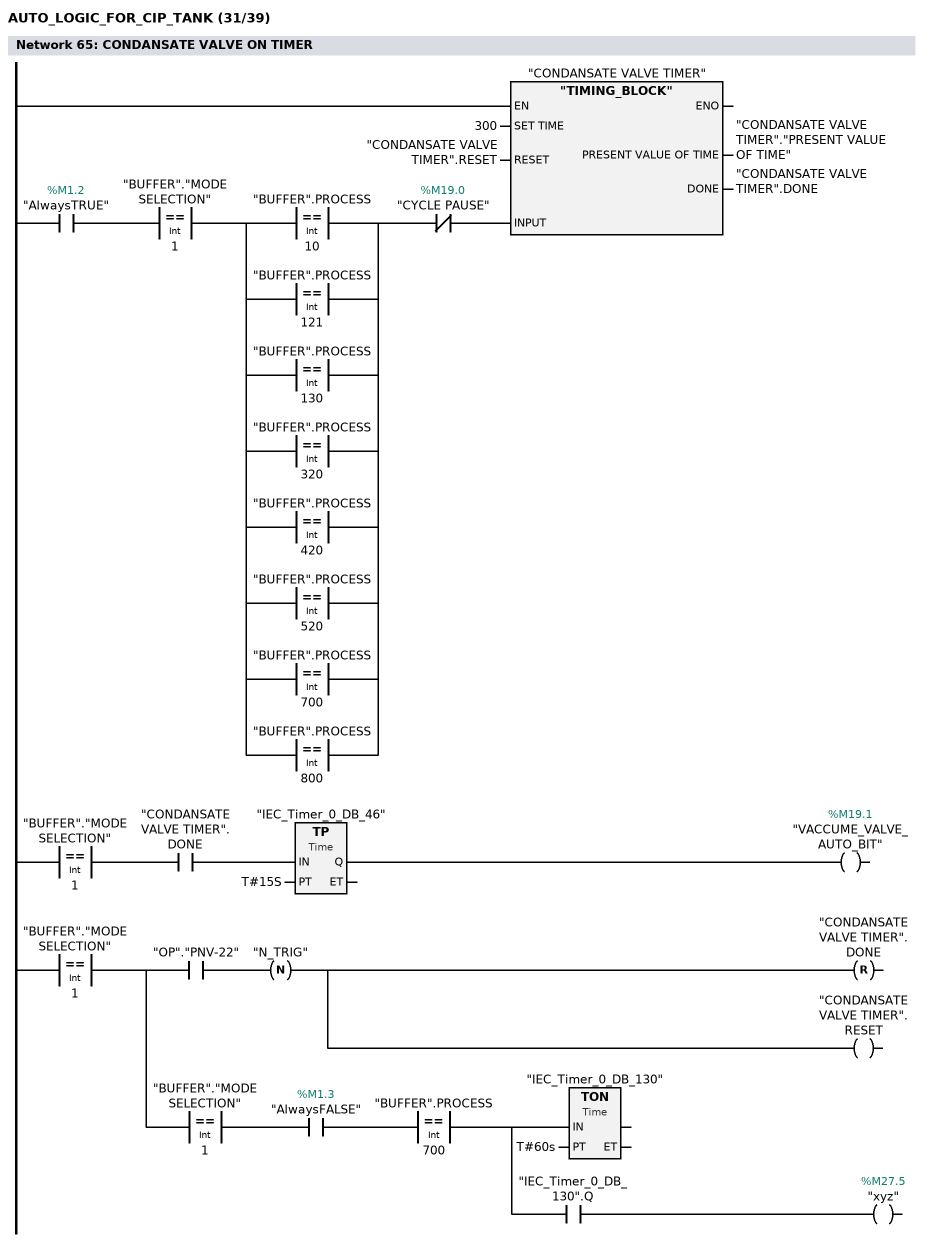
   RUNG wire#powerrail
      "CONDANSATE VALVE TIMER"(INPUT := wire#w3, "SET TIME" := 300, RESET := "CONDANSATE VALVE TIMER".RESET, "PRESENT VALUE OF TIME" => "CONDANSATE VALVE TIMER"."PRESENT VALUE OF TIME", DONE => "CONDANSATE VALVE TIMER".DONE)
   END_RUNG
   RUNG wire#powerrail
      Contact( "AlwaysTRUE" )
      { S7_Templates := "SrcType := Int" } EQ_Contact(in1 := "BUFFER"."MODE SELECTION", in2 := 1)
      wire#w1
      { S7_Templates := "SrcType := Int" } EQ_Contact(in1 := "BUFFER".PROCESS, in2 := 10)
      wire#w2
      I_Contact( "CYCLE PAUSE" )
   END_RUNG wire#w3
   RUNG wire#w1
      { S7_Templates := "SrcType := Int" } EQ_Contact(in1 := "BUFFER".PROCESS, in2 := 121)
   END_RUNG wire#w2
   RUNG wire#w1
      { S7_Templates := "SrcType := Int" } EQ_Contact(in1 := "BUFFER".PROCESS, in2 := 130)
   END_RUNG wire#w2
   RUNG wire#w1
      { S7_Templates := "SrcType := Int" } EQ_Contact(in1 := "BUFFER".PROCESS, in2 := 320)
   END_RUNG wire#w2
   RUNG wire#w1
      { S7_Templates := "SrcType := Int" } EQ_Contact(in1 := "BUFFER".PROCESS, in2 := 420)
   END_RUNG wire#w2
   RUNG wire#w1
      { S7_Templates := "SrcType := Int" } EQ_Contact(in1 := "BUFFER".PROCESS, in2 := 520)
   END_RUNG wire#w2
   RUNG wire#w1
      { S7_Templates := "SrcType := Int" } EQ_Contact(in1 := "BUFFER".PROCESS, in2 := 700)
   END_RUNG wire#w2
   RUNG wire#w1
      { S7_Templates := "SrcType := Int" } EQ_Contact(in1 := "BUFFER".PROCESS, in2 := 800)
   END_RUNG wire#w2
   RUNG wire#powerrail
      { S7_Templates := "SrcType := Int" } EQ_Contact(in1 := "BUFFER"."MODE SELECTION", in2 := 1)
      Contact( "CONDANSATE VALVE TIMER".DONE )
      { S7_Templates := "time_type := Time" } "IEC_Timer_0_DB_46".TP(pt := T#15S, et =>)
      Coil( "VACCUME_VALVE_AUTO_BIT" )
   END_RUNG
   RUNG wire#powerrail
      { S7_Templates := "SrcType := Int" } EQ_Contact(in1 := "BUFFER"."MODE SELECTION", in2 := 1)
      wire#w4
      Contact( "OP"."PNV-22" )
      N_Trig( "N_TRIG" )
      wire#w5
      R_Coil( "CONDANSATE VALVE TIMER".DONE )
   END_RUNG
   RUNG wire#w5
      Coil( "CONDANSATE VALVE TIMER".RESET )
   END_RUNG
   RUNG wire#w4
      { S7_Templates := "SrcType := Int" } EQ_Contact(in1 := "BUFFER"."MODE SELECTION", in2 := 1)
      Contact( "AlwaysFALSE" )
      { S7_Templates := "SrcType := Int" } EQ_Contact(in1 := "BUFFER".PROCESS, in2 := 700)
      wire#w6
      { S7_Templates := "time_type := Time" } "IEC_Timer_0_DB_130".TON(pt := T#60s, et =>)
   END_RUNG
   RUNG wire#w6
      Contact( "IEC_Timer_0_DB_130".Q )
      Coil( "xyz" )
   END_RUNG
   // the same network as SCL:
   "CONDANSATE VALVE TIMER"("SET TIME" := 300,   // "TIMING_BLOCK"
                           RESET := "CONDANSATE VALVE TIMER".RESET,
                           INPUT := "AlwaysTRUE" AND ("BUFFER"."MODE SELECTION" = 1) AND (("BUFFER".PROCESS = 10) OR ("BUFFER".PROCESS = 121) OR ("BUFFER".PROCESS = 130) OR ("BUFFER".PROCESS = 320) OR ("BUFFER".PROCESS = 420) OR ("BUFFER".PROCESS = 520) OR ("BUFFER".PROCESS = 700) OR ("BUFFER".PROCESS = 800)) AND NOT "CYCLE PAUSE",
                           "PRESENT VALUE OF TIME" => "CONDANSATE VALVE TIMER"."PRESENT VALUE OF TIME",
                           DONE => "CONDANSATE VALVE TIMER".DONE);
   "IEC_Timer_0_DB_46".TP(IN := ("BUFFER"."MODE SELECTION" = 1) AND "CONDANSATE VALVE TIMER".DONE, PT := T#15S);
   "VACCUME_VALVE_AUTO_BIT" := "IEC_Timer_0_DB_46".Q;
   #_w1 := "BUFFER"."MODE SELECTION" = 1;
   #_w2 := #_w1 AND "OP"."PNV-22";
   #_w3 := NOT #_w2 AND "N_TRIG";   // falling edge
   "N_TRIG" := #_w2;
   IF #_w3 THEN "CONDANSATE VALVE TIMER".DONE := FALSE; END_IF;
   "CONDANSATE VALVE TIMER".RESET := #_w3;
   #_w4 := #_w1 AND ("BUFFER"."MODE SELECTION" = 1) AND "AlwaysFALSE" AND ("BUFFER".PROCESS = 700);
   "IEC_Timer_0_DB_130".TON(IN := #_w4, PT := T#60s);
   "xyz" := #_w4 AND "IEC_Timer_0_DB_130".Q;
END_REGION

REGION Network 68: -----------------SELF CLEANING CIP TANK---------------------- NEW LOGIC ADD
END_REGION

REGION Network 69: START SW TANK
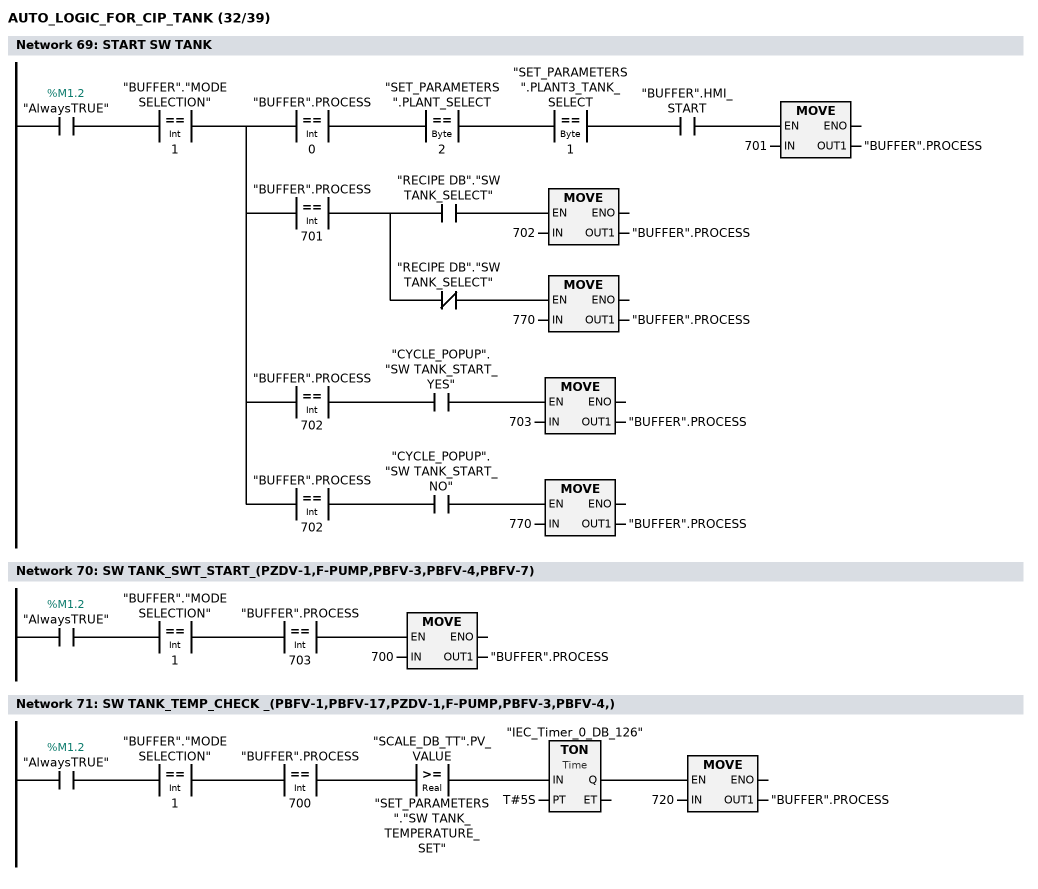
   RUNG wire#powerrail
      Contact( "AlwaysTRUE" )
      { S7_Templates := "SrcType := Int" } EQ_Contact(in1 := "BUFFER"."MODE SELECTION", in2 := 1)
      wire#w1
      { S7_Templates := "SrcType := Int" } EQ_Contact(in1 := "BUFFER".PROCESS, in2 := 0)
      { S7_Templates := "SrcType := Byte" } EQ_Contact(in1 := "SET_PARAMETERS".PLANT_SELECT, in2 := 2)
      { S7_Templates := "SrcType := Byte" } EQ_Contact(in1 := "SET_PARAMETERS".PLANT3_TANK_SELECT, in2 := 1)
      Contact( "BUFFER".HMI_START )
      Move(in := 701, out1 => "BUFFER".PROCESS)
   END_RUNG
   RUNG wire#w1
      { S7_Templates := "SrcType := Int" } EQ_Contact(in1 := "BUFFER".PROCESS, in2 := 701)
      wire#w2
      Contact( "RECIPE DB"."SW TANK_SELECT" )
      Move(in := 702, out1 => "BUFFER".PROCESS)
   END_RUNG
   RUNG wire#w2
      I_Contact( "RECIPE DB"."SW TANK_SELECT" )
      Move(in := 770, out1 => "BUFFER".PROCESS)
   END_RUNG
   RUNG wire#w1
      { S7_Templates := "SrcType := Int" } EQ_Contact(in1 := "BUFFER".PROCESS, in2 := 702)
      Contact( "CYCLE_POPUP"."SW TANK_START_YES" )
      Move(in := 703, out1 => "BUFFER".PROCESS)
   END_RUNG
   RUNG wire#w1
      { S7_Templates := "SrcType := Int" } EQ_Contact(in1 := "BUFFER".PROCESS, in2 := 702)
      Contact( "CYCLE_POPUP"."SW TANK_START_NO" )
      Move(in := 770, out1 => "BUFFER".PROCESS)
   END_RUNG
   // the same network as SCL:
   #_w1 := "AlwaysTRUE" AND ("BUFFER"."MODE SELECTION" = 1);
   IF #_w1 AND ("BUFFER".PROCESS = 0) AND ("SET_PARAMETERS".PLANT_SELECT = 2) AND ("SET_PARAMETERS".PLANT3_TANK_SELECT = 1) AND "BUFFER".HMI_START THEN
       "BUFFER".PROCESS := 701;
   END_IF;
   #_w2 := #_w1 AND ("BUFFER".PROCESS = 701);
   IF #_w2 AND "RECIPE DB"."SW TANK_SELECT" THEN "BUFFER".PROCESS := 702; END_IF;
   IF #_w2 AND NOT "RECIPE DB"."SW TANK_SELECT" THEN "BUFFER".PROCESS := 770; END_IF;
   IF #_w1 AND ("BUFFER".PROCESS = 702) AND "CYCLE_POPUP"."SW TANK_START_YES" THEN
       "BUFFER".PROCESS := 703;
   END_IF;
   IF #_w1 AND ("BUFFER".PROCESS = 702) AND "CYCLE_POPUP"."SW TANK_START_NO" THEN
       "BUFFER".PROCESS := 770;
   END_IF;
END_REGION

REGION Network 70: SW TANK_SWT_START_(PZDV-1,F-PUMP,PBFV-3,PBFV-4,PBFV-7)
   RUNG wire#powerrail
      Contact( "AlwaysTRUE" )
      { S7_Templates := "SrcType := Int" } EQ_Contact(in1 := "BUFFER"."MODE SELECTION", in2 := 1)
      { S7_Templates := "SrcType := Int" } EQ_Contact(in1 := "BUFFER".PROCESS, in2 := 703)
      Move(in := 700, out1 => "BUFFER".PROCESS)
   END_RUNG
   // the same network as SCL:
   IF "AlwaysTRUE" AND ("BUFFER"."MODE SELECTION" = 1) AND ("BUFFER".PROCESS = 703) THEN
       "BUFFER".PROCESS := 700;
   END_IF;
END_REGION

REGION Network 71: SW TANK_TEMP_CHECK _(PBFV-1,PBFV-17,PZDV-1,F-PUMP,PBFV-3,PBFV-4,)
   RUNG wire#powerrail
      Contact( "AlwaysTRUE" )
      { S7_Templates := "SrcType := Int" } EQ_Contact(in1 := "BUFFER"."MODE SELECTION", in2 := 1)
      { S7_Templates := "SrcType := Int" } EQ_Contact(in1 := "BUFFER".PROCESS, in2 := 700)
      { S7_Templates := "SrcType := Real" } GE_Contact(in1 := "SCALE_DB_TT".PV_VALUE, in2 := "SET_PARAMETERS"."SW TANK_TEMPERATURE_SET")
      { S7_Templates := "time_type := Time" } "IEC_Timer_0_DB_126".TON(pt := T#5S, et =>)
      Move(in := 720, out1 => "BUFFER".PROCESS)
   END_RUNG
   // the same network as SCL:
   "IEC_Timer_0_DB_126".TON(IN := "AlwaysTRUE" AND ("BUFFER"."MODE SELECTION" = 1) AND ("BUFFER".PROCESS = 700) AND ("SCALE_DB_TT".PV_VALUE >= "SET_PARAMETERS"."SW TANK_TEMPERATURE_SET"),
                           PT := T#5S);
   IF "IEC_Timer_0_DB_126".Q THEN "BUFFER".PROCESS := 720; END_IF;
END_REGION

REGION Network 72: SW TANK_CLEANING_TIME_(PZDV-1,F-PUMP,PBFV-3,PBFV-4)
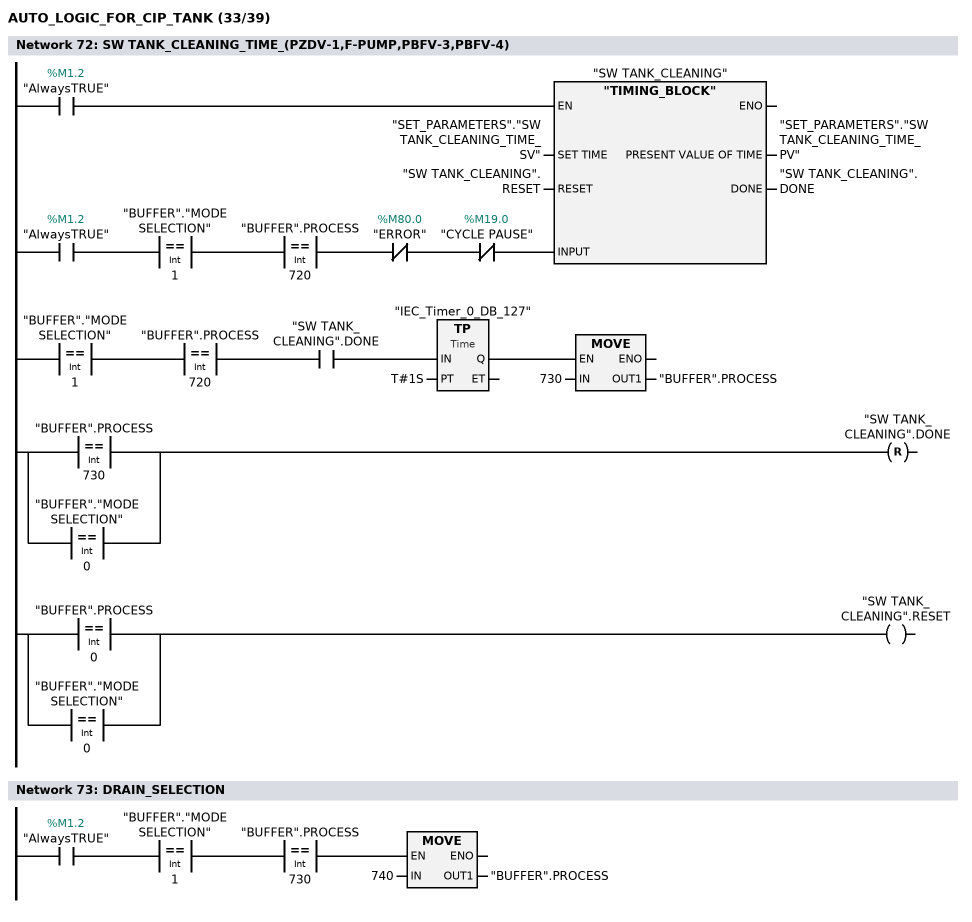
   RUNG wire#powerrail
      Contact( "AlwaysTRUE" )
      "SW TANK_CLEANING"(INPUT := wire#w1, "SET TIME" := "SET_PARAMETERS"."SW TANK_CLEANING_TIME_SV", RESET := "SW TANK_CLEANING".RESET, "PRESENT VALUE OF TIME" => "SET_PARAMETERS"."SW TANK_CLEANING_TIME_PV", DONE => "SW TANK_CLEANING".DONE)
   END_RUNG
   RUNG wire#powerrail
      Contact( "AlwaysTRUE" )
      { S7_Templates := "SrcType := Int" } EQ_Contact(in1 := "BUFFER"."MODE SELECTION", in2 := 1)
      { S7_Templates := "SrcType := Int" } EQ_Contact(in1 := "BUFFER".PROCESS, in2 := 720)
      I_Contact( "ERROR" )
      I_Contact( "CYCLE PAUSE" )
   END_RUNG wire#w1
   RUNG wire#powerrail
      { S7_Templates := "SrcType := Int" } EQ_Contact(in1 := "BUFFER"."MODE SELECTION", in2 := 1)
      { S7_Templates := "SrcType := Int" } EQ_Contact(in1 := "BUFFER".PROCESS, in2 := 720)
      Contact( "SW TANK_CLEANING".DONE )
      { S7_Templates := "time_type := Time" } "IEC_Timer_0_DB_127".TP(pt := T#1S, et =>)
      Move(in := 730, out1 => "BUFFER".PROCESS)
   END_RUNG
   RUNG wire#powerrail
      { S7_Templates := "SrcType := Int" } EQ_Contact(in1 := "BUFFER".PROCESS, in2 := 730)
      wire#w2
      R_Coil( "SW TANK_CLEANING".DONE )
   END_RUNG
   RUNG wire#powerrail
      { S7_Templates := "SrcType := Int" } EQ_Contact(in1 := "BUFFER"."MODE SELECTION", in2 := 0)
   END_RUNG wire#w2
   RUNG wire#powerrail
      { S7_Templates := "SrcType := Int" } EQ_Contact(in1 := "BUFFER".PROCESS, in2 := 0)
      wire#w3
      Coil( "SW TANK_CLEANING".RESET )
   END_RUNG
   RUNG wire#powerrail
      { S7_Templates := "SrcType := Int" } EQ_Contact(in1 := "BUFFER"."MODE SELECTION", in2 := 0)
   END_RUNG wire#w3
   // the same network as SCL:
   IF "AlwaysTRUE" THEN
       "SW TANK_CLEANING"("SET TIME" := "SET_PARAMETERS"."SW TANK_CLEANING_TIME_SV",   // "TIMING_BLOCK"
                          RESET := "SW TANK_CLEANING".RESET,
                          INPUT := "AlwaysTRUE" AND ("BUFFER"."MODE SELECTION" = 1) AND ("BUFFER".PROCESS = 720) AND NOT "ERROR" AND NOT "CYCLE PAUSE",
                          "PRESENT VALUE OF TIME" => "SET_PARAMETERS"."SW TANK_CLEANING_TIME_PV",
                          DONE => "SW TANK_CLEANING".DONE);
   END_IF;
   "IEC_Timer_0_DB_127".TP(IN := ("BUFFER"."MODE SELECTION" = 1) AND ("BUFFER".PROCESS = 720) AND "SW TANK_CLEANING".DONE,
                           PT := T#1S);
   IF "IEC_Timer_0_DB_127".Q THEN "BUFFER".PROCESS := 730; END_IF;
   IF ("BUFFER".PROCESS = 730) OR ("BUFFER"."MODE SELECTION" = 0) THEN
       "SW TANK_CLEANING".DONE := FALSE;
   END_IF;
   "SW TANK_CLEANING".RESET := ("BUFFER".PROCESS = 0) OR ("BUFFER"."MODE SELECTION" = 0);
END_REGION

REGION Network 73: DRAIN_SELECTION
   RUNG wire#powerrail
      Contact( "AlwaysTRUE" )
      { S7_Templates := "SrcType := Int" } EQ_Contact(in1 := "BUFFER"."MODE SELECTION", in2 := 1)
      { S7_Templates := "SrcType := Int" } EQ_Contact(in1 := "BUFFER".PROCESS, in2 := 730)
      Move(in := 740, out1 => "BUFFER".PROCESS)
   END_RUNG
   // the same network as SCL:
   IF "AlwaysTRUE" AND ("BUFFER"."MODE SELECTION" = 1) AND ("BUFFER".PROCESS = 730) THEN
       "BUFFER".PROCESS := 740;
   END_IF;
END_REGION

REGION Network 74: SW TANK_DRAIN_TIME_(PZDV-1,F PUMP,PBFV-5,PBFV-6,PBFV-11) PRACTICAL
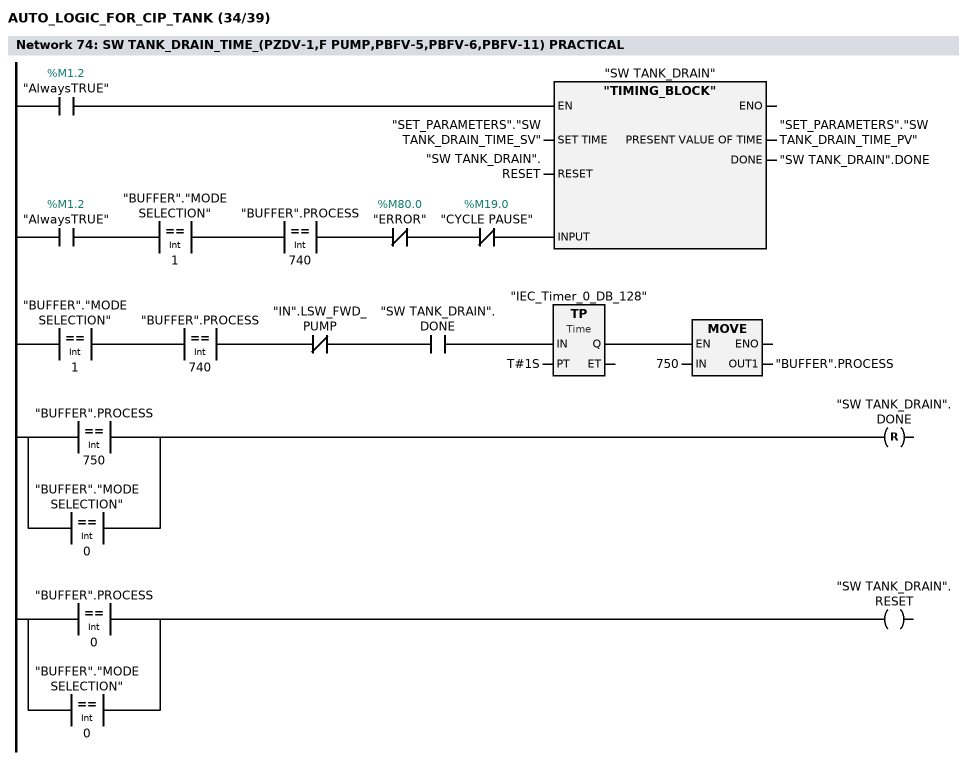
   RUNG wire#powerrail
      Contact( "AlwaysTRUE" )
      "SW TANK_DRAIN"(INPUT := wire#w1, "SET TIME" := "SET_PARAMETERS"."SW TANK_DRAIN_TIME_SV", RESET := "SW TANK_DRAIN".RESET, "PRESENT VALUE OF TIME" => "SET_PARAMETERS"."SW TANK_DRAIN_TIME_PV", DONE => "SW TANK_DRAIN".DONE)
   END_RUNG
   RUNG wire#powerrail
      Contact( "AlwaysTRUE" )
      { S7_Templates := "SrcType := Int" } EQ_Contact(in1 := "BUFFER"."MODE SELECTION", in2 := 1)
      { S7_Templates := "SrcType := Int" } EQ_Contact(in1 := "BUFFER".PROCESS, in2 := 740)
      I_Contact( "ERROR" )
      I_Contact( "CYCLE PAUSE" )
   END_RUNG wire#w1
   RUNG wire#powerrail
      { S7_Templates := "SrcType := Int" } EQ_Contact(in1 := "BUFFER"."MODE SELECTION", in2 := 1)
      { S7_Templates := "SrcType := Int" } EQ_Contact(in1 := "BUFFER".PROCESS, in2 := 740)
      I_Contact( "IN".LSW_FWD_PUMP )
      Contact( "SW TANK_DRAIN".DONE )
      { S7_Templates := "time_type := Time" } "IEC_Timer_0_DB_128".TP(pt := T#1S, et =>)
      Move(in := 750, out1 => "BUFFER".PROCESS)
   END_RUNG
   RUNG wire#powerrail
      { S7_Templates := "SrcType := Int" } EQ_Contact(in1 := "BUFFER".PROCESS, in2 := 750)
      wire#w2
      R_Coil( "SW TANK_DRAIN".DONE )
   END_RUNG
   RUNG wire#powerrail
      { S7_Templates := "SrcType := Int" } EQ_Contact(in1 := "BUFFER"."MODE SELECTION", in2 := 0)
   END_RUNG wire#w2
   RUNG wire#powerrail
      { S7_Templates := "SrcType := Int" } EQ_Contact(in1 := "BUFFER".PROCESS, in2 := 0)
      wire#w3
      Coil( "SW TANK_DRAIN".RESET )
   END_RUNG
   RUNG wire#powerrail
      { S7_Templates := "SrcType := Int" } EQ_Contact(in1 := "BUFFER"."MODE SELECTION", in2 := 0)
   END_RUNG wire#w3
   // the same network as SCL:
   IF "AlwaysTRUE" THEN
       "SW TANK_DRAIN"("SET TIME" := "SET_PARAMETERS"."SW TANK_DRAIN_TIME_SV",   // "TIMING_BLOCK"
                       RESET := "SW TANK_DRAIN".RESET,
                       INPUT := "AlwaysTRUE" AND ("BUFFER"."MODE SELECTION" = 1) AND ("BUFFER".PROCESS = 740) AND NOT "ERROR" AND NOT "CYCLE PAUSE",
                       "PRESENT VALUE OF TIME" => "SET_PARAMETERS"."SW TANK_DRAIN_TIME_PV",
                       DONE => "SW TANK_DRAIN".DONE);
   END_IF;
   "IEC_Timer_0_DB_128".TP(IN := ("BUFFER"."MODE SELECTION" = 1) AND ("BUFFER".PROCESS = 740) AND NOT "IN".LSW_FWD_PUMP AND "SW TANK_DRAIN".DONE,
                           PT := T#1S);
   IF "IEC_Timer_0_DB_128".Q THEN "BUFFER".PROCESS := 750; END_IF;
   IF ("BUFFER".PROCESS = 750) OR ("BUFFER"."MODE SELECTION" = 0) THEN "SW TANK_DRAIN".DONE := FALSE; END_IF;
   "SW TANK_DRAIN".RESET := ("BUFFER".PROCESS = 0) OR ("BUFFER"."MODE SELECTION" = 0);
END_REGION

REGION Network 75: SW TANK_PUMP_CHASING_TIME(PBFV-12,PBFV13) FAKE TYPE AUDIT NOT OPERATE OUTPUT
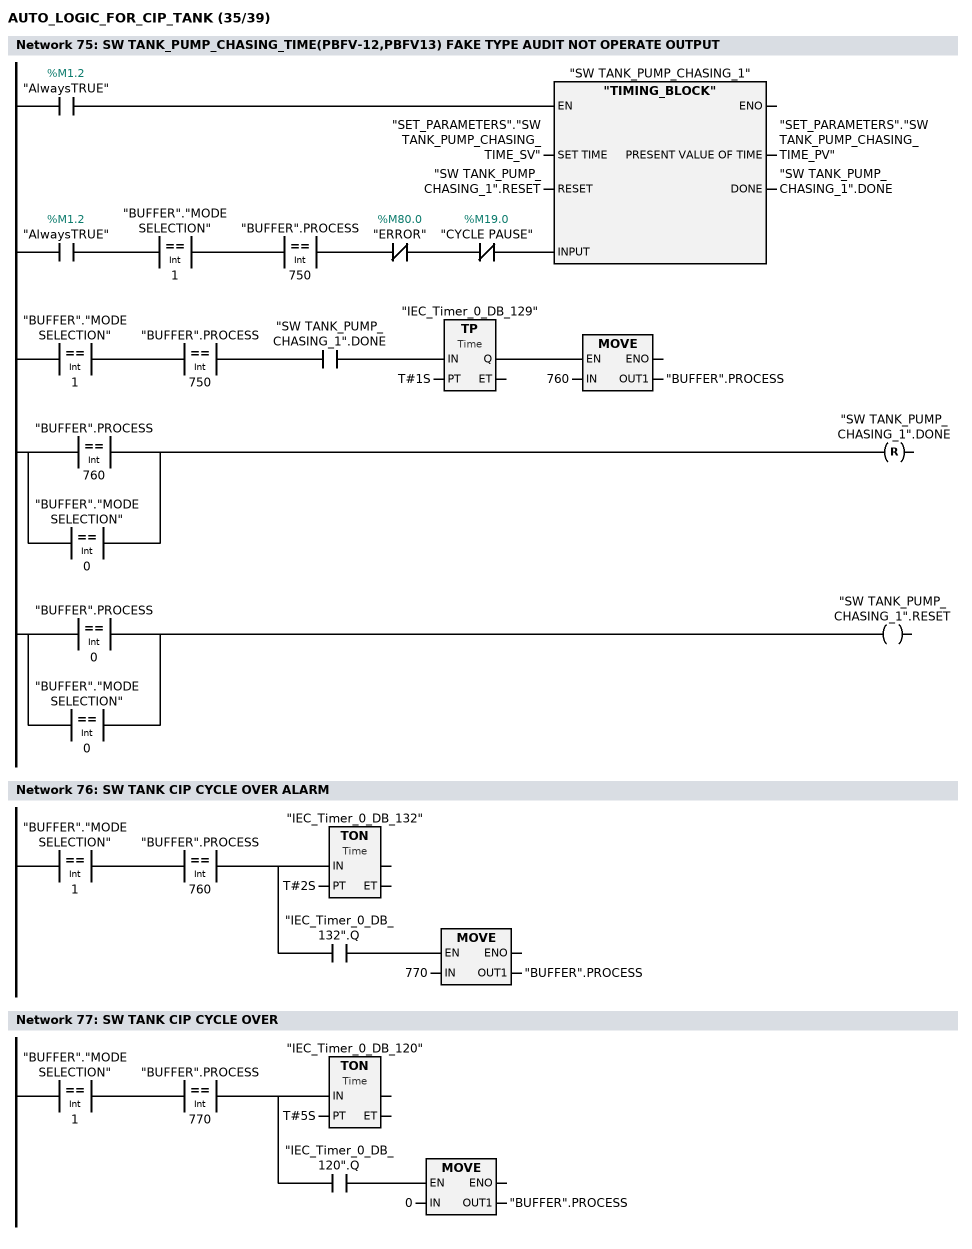
   RUNG wire#powerrail
      Contact( "AlwaysTRUE" )
      "SW TANK_PUMP_CHASING_1"(INPUT := wire#w1, "SET TIME" := "SET_PARAMETERS"."SW TANK_PUMP_CHASING_TIME_SV", RESET := "SW TANK_PUMP_CHASING_1".RESET, "PRESENT VALUE OF TIME" => "SET_PARAMETERS"."SW TANK_PUMP_CHASING_TIME_PV", DONE => "SW TANK_PUMP_CHASING_1".DONE)
   END_RUNG
   RUNG wire#powerrail
      Contact( "AlwaysTRUE" )
      { S7_Templates := "SrcType := Int" } EQ_Contact(in1 := "BUFFER"."MODE SELECTION", in2 := 1)
      { S7_Templates := "SrcType := Int" } EQ_Contact(in1 := "BUFFER".PROCESS, in2 := 750)
      I_Contact( "ERROR" )
      I_Contact( "CYCLE PAUSE" )
   END_RUNG wire#w1
   RUNG wire#powerrail
      { S7_Templates := "SrcType := Int" } EQ_Contact(in1 := "BUFFER"."MODE SELECTION", in2 := 1)
      { S7_Templates := "SrcType := Int" } EQ_Contact(in1 := "BUFFER".PROCESS, in2 := 750)
      Contact( "SW TANK_PUMP_CHASING_1".DONE )
      { S7_Templates := "time_type := Time" } "IEC_Timer_0_DB_129".TP(pt := T#1S, et =>)
      Move(in := 760, out1 => "BUFFER".PROCESS)
   END_RUNG
   RUNG wire#powerrail
      { S7_Templates := "SrcType := Int" } EQ_Contact(in1 := "BUFFER".PROCESS, in2 := 760)
      wire#w2
      R_Coil( "SW TANK_PUMP_CHASING_1".DONE )
   END_RUNG
   RUNG wire#powerrail
      { S7_Templates := "SrcType := Int" } EQ_Contact(in1 := "BUFFER"."MODE SELECTION", in2 := 0)
   END_RUNG wire#w2
   RUNG wire#powerrail
      { S7_Templates := "SrcType := Int" } EQ_Contact(in1 := "BUFFER".PROCESS, in2 := 0)
      wire#w3
      Coil( "SW TANK_PUMP_CHASING_1".RESET )
   END_RUNG
   RUNG wire#powerrail
      { S7_Templates := "SrcType := Int" } EQ_Contact(in1 := "BUFFER"."MODE SELECTION", in2 := 0)
   END_RUNG wire#w3
   // the same network as SCL:
   IF "AlwaysTRUE" THEN
       "SW TANK_PUMP_CHASING_1"("SET TIME" := "SET_PARAMETERS"."SW TANK_PUMP_CHASING_TIME_SV",   // "TIMING_BLOCK"
                               RESET := "SW TANK_PUMP_CHASING_1".RESET,
                               INPUT := "AlwaysTRUE" AND ("BUFFER"."MODE SELECTION" = 1) AND ("BUFFER".PROCESS = 750) AND NOT "ERROR" AND NOT "CYCLE PAUSE",
                               "PRESENT VALUE OF TIME" => "SET_PARAMETERS"."SW TANK_PUMP_CHASING_TIME_PV",
                               DONE => "SW TANK_PUMP_CHASING_1".DONE);
   END_IF;
   "IEC_Timer_0_DB_129".TP(IN := ("BUFFER"."MODE SELECTION" = 1) AND ("BUFFER".PROCESS = 750) AND "SW TANK_PUMP_CHASING_1".DONE,
                           PT := T#1S);
   IF "IEC_Timer_0_DB_129".Q THEN "BUFFER".PROCESS := 760; END_IF;
   IF ("BUFFER".PROCESS = 760) OR ("BUFFER"."MODE SELECTION" = 0) THEN
       "SW TANK_PUMP_CHASING_1".DONE := FALSE;
   END_IF;
   "SW TANK_PUMP_CHASING_1".RESET := ("BUFFER".PROCESS = 0) OR ("BUFFER"."MODE SELECTION" = 0);
END_REGION

REGION Network 76: SW TANK CIP CYCLE OVER ALARM
   RUNG wire#powerrail
      { S7_Templates := "SrcType := Int" } EQ_Contact(in1 := "BUFFER"."MODE SELECTION", in2 := 1)
      { S7_Templates := "SrcType := Int" } EQ_Contact(in1 := "BUFFER".PROCESS, in2 := 760)
      wire#w1
      { S7_Templates := "time_type := Time" } "IEC_Timer_0_DB_132".TON(pt := T#2S, et =>)
   END_RUNG
   RUNG wire#w1
      Contact( "IEC_Timer_0_DB_132".Q )
      Move(in := 770, out1 => "BUFFER".PROCESS)
   END_RUNG
   // the same network as SCL:
   #_w1 := ("BUFFER"."MODE SELECTION" = 1) AND ("BUFFER".PROCESS = 760);
   "IEC_Timer_0_DB_132".TON(IN := #_w1, PT := T#2S);
   IF #_w1 AND "IEC_Timer_0_DB_132".Q THEN "BUFFER".PROCESS := 770; END_IF;
END_REGION

REGION Network 77: SW TANK CIP CYCLE OVER
   RUNG wire#powerrail
      { S7_Templates := "SrcType := Int" } EQ_Contact(in1 := "BUFFER"."MODE SELECTION", in2 := 1)
      { S7_Templates := "SrcType := Int" } EQ_Contact(in1 := "BUFFER".PROCESS, in2 := 770)
      wire#w1
      { S7_Templates := "time_type := Time" } "IEC_Timer_0_DB_120".TON(pt := T#5S, et =>)
   END_RUNG
   RUNG wire#w1
      Contact( "IEC_Timer_0_DB_120".Q )
      Move(in := 0, out1 => "BUFFER".PROCESS)
   END_RUNG
   // the same network as SCL:
   #_w1 := ("BUFFER"."MODE SELECTION" = 1) AND ("BUFFER".PROCESS = 770);
   "IEC_Timer_0_DB_120".TON(IN := #_w1, PT := T#5S);
   IF #_w1 AND "IEC_Timer_0_DB_120".Q THEN "BUFFER".PROCESS := 0; END_IF;
END_REGION

REGION Network 79: START PW TANK
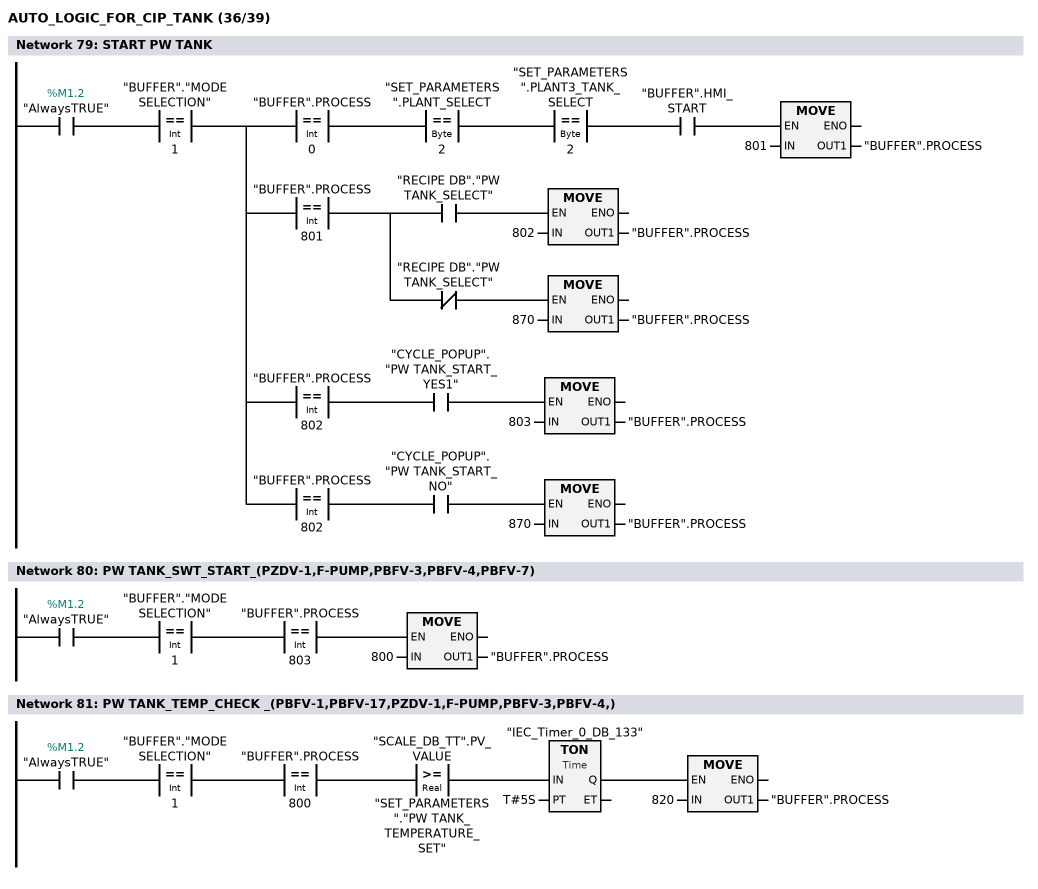
   RUNG wire#powerrail
      Contact( "AlwaysTRUE" )
      { S7_Templates := "SrcType := Int" } EQ_Contact(in1 := "BUFFER"."MODE SELECTION", in2 := 1)
      wire#w1
      { S7_Templates := "SrcType := Int" } EQ_Contact(in1 := "BUFFER".PROCESS, in2 := 0)
      { S7_Templates := "SrcType := Byte" } EQ_Contact(in1 := "SET_PARAMETERS".PLANT_SELECT, in2 := 2)
      { S7_Templates := "SrcType := Byte" } EQ_Contact(in1 := "SET_PARAMETERS".PLANT3_TANK_SELECT, in2 := 2)
      Contact( "BUFFER".HMI_START )
      Move(in := 801, out1 => "BUFFER".PROCESS)
   END_RUNG
   RUNG wire#w1
      { S7_Templates := "SrcType := Int" } EQ_Contact(in1 := "BUFFER".PROCESS, in2 := 801)
      wire#w2
      Contact( "RECIPE DB"."PW TANK_SELECT" )
      Move(in := 802, out1 => "BUFFER".PROCESS)
   END_RUNG
   RUNG wire#w2
      I_Contact( "RECIPE DB"."PW TANK_SELECT" )
      Move(in := 870, out1 => "BUFFER".PROCESS)
   END_RUNG
   RUNG wire#w1
      { S7_Templates := "SrcType := Int" } EQ_Contact(in1 := "BUFFER".PROCESS, in2 := 802)
      Contact( "CYCLE_POPUP"."PW TANK_START_YES1" )
      Move(in := 803, out1 => "BUFFER".PROCESS)
   END_RUNG
   RUNG wire#w1
      { S7_Templates := "SrcType := Int" } EQ_Contact(in1 := "BUFFER".PROCESS, in2 := 802)
      Contact( "CYCLE_POPUP"."PW TANK_START_NO" )
      Move(in := 870, out1 => "BUFFER".PROCESS)
   END_RUNG
   // the same network as SCL:
   #_w1 := "AlwaysTRUE" AND ("BUFFER"."MODE SELECTION" = 1);
   IF #_w1 AND ("BUFFER".PROCESS = 0) AND ("SET_PARAMETERS".PLANT_SELECT = 2) AND ("SET_PARAMETERS".PLANT3_TANK_SELECT = 2) AND "BUFFER".HMI_START THEN
       "BUFFER".PROCESS := 801;
   END_IF;
   #_w2 := #_w1 AND ("BUFFER".PROCESS = 801);
   IF #_w2 AND "RECIPE DB"."PW TANK_SELECT" THEN "BUFFER".PROCESS := 802; END_IF;
   IF #_w2 AND NOT "RECIPE DB"."PW TANK_SELECT" THEN "BUFFER".PROCESS := 870; END_IF;
   IF #_w1 AND ("BUFFER".PROCESS = 802) AND "CYCLE_POPUP"."PW TANK_START_YES1" THEN
       "BUFFER".PROCESS := 803;
   END_IF;
   IF #_w1 AND ("BUFFER".PROCESS = 802) AND "CYCLE_POPUP"."PW TANK_START_NO" THEN
       "BUFFER".PROCESS := 870;
   END_IF;
END_REGION

REGION Network 80: PW TANK_SWT_START_(PZDV-1,F-PUMP,PBFV-3,PBFV-4,PBFV-7)
   RUNG wire#powerrail
      Contact( "AlwaysTRUE" )
      { S7_Templates := "SrcType := Int" } EQ_Contact(in1 := "BUFFER"."MODE SELECTION", in2 := 1)
      { S7_Templates := "SrcType := Int" } EQ_Contact(in1 := "BUFFER".PROCESS, in2 := 803)
      Move(in := 800, out1 => "BUFFER".PROCESS)
   END_RUNG
   // the same network as SCL:
   IF "AlwaysTRUE" AND ("BUFFER"."MODE SELECTION" = 1) AND ("BUFFER".PROCESS = 803) THEN
       "BUFFER".PROCESS := 800;
   END_IF;
END_REGION

REGION Network 81: PW TANK_TEMP_CHECK _(PBFV-1,PBFV-17,PZDV-1,F-PUMP,PBFV-3,PBFV-4,)
   RUNG wire#powerrail
      Contact( "AlwaysTRUE" )
      { S7_Templates := "SrcType := Int" } EQ_Contact(in1 := "BUFFER"."MODE SELECTION", in2 := 1)
      { S7_Templates := "SrcType := Int" } EQ_Contact(in1 := "BUFFER".PROCESS, in2 := 800)
      { S7_Templates := "SrcType := Real" } GE_Contact(in1 := "SCALE_DB_TT".PV_VALUE, in2 := "SET_PARAMETERS"."PW TANK_TEMPERATURE_SET")
      { S7_Templates := "time_type := Time" } "IEC_Timer_0_DB_133".TON(pt := T#5S, et =>)
      Move(in := 820, out1 => "BUFFER".PROCESS)
   END_RUNG
   // the same network as SCL:
   "IEC_Timer_0_DB_133".TON(IN := "AlwaysTRUE" AND ("BUFFER"."MODE SELECTION" = 1) AND ("BUFFER".PROCESS = 800) AND ("SCALE_DB_TT".PV_VALUE >= "SET_PARAMETERS"."PW TANK_TEMPERATURE_SET"),
                           PT := T#5S);
   IF "IEC_Timer_0_DB_133".Q THEN "BUFFER".PROCESS := 820; END_IF;
END_REGION

REGION Network 82: PW TANK_CLEANING_TIME_(PZDV-1,F-PUMP,PBFV-3,PBFV-4)
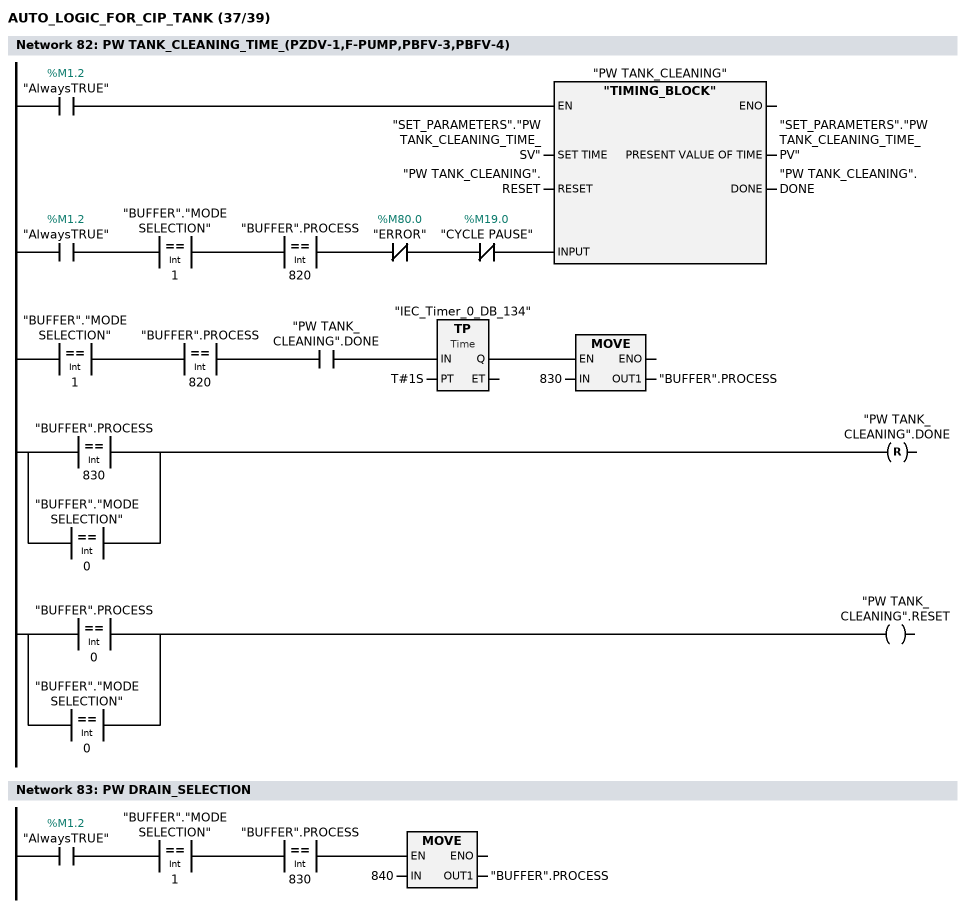
   RUNG wire#powerrail
      Contact( "AlwaysTRUE" )
      "PW TANK_CLEANING"(INPUT := wire#w1, "SET TIME" := "SET_PARAMETERS"."PW TANK_CLEANING_TIME_SV", RESET := "PW TANK_CLEANING".RESET, "PRESENT VALUE OF TIME" => "SET_PARAMETERS"."PW TANK_CLEANING_TIME_PV", DONE => "PW TANK_CLEANING".DONE)
   END_RUNG
   RUNG wire#powerrail
      Contact( "AlwaysTRUE" )
      { S7_Templates := "SrcType := Int" } EQ_Contact(in1 := "BUFFER"."MODE SELECTION", in2 := 1)
      { S7_Templates := "SrcType := Int" } EQ_Contact(in1 := "BUFFER".PROCESS, in2 := 820)
      I_Contact( "ERROR" )
      I_Contact( "CYCLE PAUSE" )
   END_RUNG wire#w1
   RUNG wire#powerrail
      { S7_Templates := "SrcType := Int" } EQ_Contact(in1 := "BUFFER"."MODE SELECTION", in2 := 1)
      { S7_Templates := "SrcType := Int" } EQ_Contact(in1 := "BUFFER".PROCESS, in2 := 820)
      Contact( "PW TANK_CLEANING".DONE )
      { S7_Templates := "time_type := Time" } "IEC_Timer_0_DB_134".TP(pt := T#1S, et =>)
      Move(in := 830, out1 => "BUFFER".PROCESS)
   END_RUNG
   RUNG wire#powerrail
      { S7_Templates := "SrcType := Int" } EQ_Contact(in1 := "BUFFER".PROCESS, in2 := 830)
      wire#w2
      R_Coil( "PW TANK_CLEANING".DONE )
   END_RUNG
   RUNG wire#powerrail
      { S7_Templates := "SrcType := Int" } EQ_Contact(in1 := "BUFFER"."MODE SELECTION", in2 := 0)
   END_RUNG wire#w2
   RUNG wire#powerrail
      { S7_Templates := "SrcType := Int" } EQ_Contact(in1 := "BUFFER".PROCESS, in2 := 0)
      wire#w3
      Coil( "PW TANK_CLEANING".RESET )
   END_RUNG
   RUNG wire#powerrail
      { S7_Templates := "SrcType := Int" } EQ_Contact(in1 := "BUFFER"."MODE SELECTION", in2 := 0)
   END_RUNG wire#w3
   // the same network as SCL:
   IF "AlwaysTRUE" THEN
       "PW TANK_CLEANING"("SET TIME" := "SET_PARAMETERS"."PW TANK_CLEANING_TIME_SV",   // "TIMING_BLOCK"
                          RESET := "PW TANK_CLEANING".RESET,
                          INPUT := "AlwaysTRUE" AND ("BUFFER"."MODE SELECTION" = 1) AND ("BUFFER".PROCESS = 820) AND NOT "ERROR" AND NOT "CYCLE PAUSE",
                          "PRESENT VALUE OF TIME" => "SET_PARAMETERS"."PW TANK_CLEANING_TIME_PV",
                          DONE => "PW TANK_CLEANING".DONE);
   END_IF;
   "IEC_Timer_0_DB_134".TP(IN := ("BUFFER"."MODE SELECTION" = 1) AND ("BUFFER".PROCESS = 820) AND "PW TANK_CLEANING".DONE,
                           PT := T#1S);
   IF "IEC_Timer_0_DB_134".Q THEN "BUFFER".PROCESS := 830; END_IF;
   IF ("BUFFER".PROCESS = 830) OR ("BUFFER"."MODE SELECTION" = 0) THEN
       "PW TANK_CLEANING".DONE := FALSE;
   END_IF;
   "PW TANK_CLEANING".RESET := ("BUFFER".PROCESS = 0) OR ("BUFFER"."MODE SELECTION" = 0);
END_REGION

REGION Network 83: PW DRAIN_SELECTION
   RUNG wire#powerrail
      Contact( "AlwaysTRUE" )
      { S7_Templates := "SrcType := Int" } EQ_Contact(in1 := "BUFFER"."MODE SELECTION", in2 := 1)
      { S7_Templates := "SrcType := Int" } EQ_Contact(in1 := "BUFFER".PROCESS, in2 := 830)
      Move(in := 840, out1 => "BUFFER".PROCESS)
   END_RUNG
   // the same network as SCL:
   IF "AlwaysTRUE" AND ("BUFFER"."MODE SELECTION" = 1) AND ("BUFFER".PROCESS = 830) THEN
       "BUFFER".PROCESS := 840;
   END_IF;
END_REGION

REGION Network 84: PW TANK_DRAIN_TIME_(PZDV-1,F PUMP,PBFV-5,PBFV-6,PBFV-11) PRACTICAL
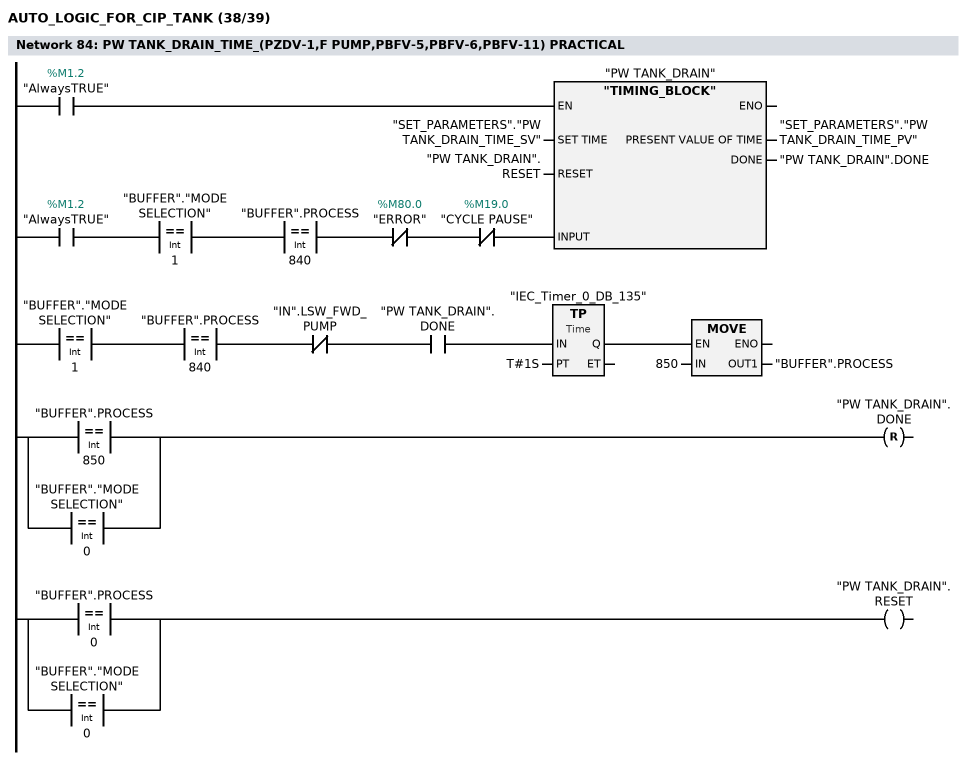
   RUNG wire#powerrail
      Contact( "AlwaysTRUE" )
      "PW TANK_DRAIN"(INPUT := wire#w1, "SET TIME" := "SET_PARAMETERS"."PW TANK_DRAIN_TIME_SV", RESET := "PW TANK_DRAIN".RESET, "PRESENT VALUE OF TIME" => "SET_PARAMETERS"."PW TANK_DRAIN_TIME_PV", DONE => "PW TANK_DRAIN".DONE)
   END_RUNG
   RUNG wire#powerrail
      Contact( "AlwaysTRUE" )
      { S7_Templates := "SrcType := Int" } EQ_Contact(in1 := "BUFFER"."MODE SELECTION", in2 := 1)
      { S7_Templates := "SrcType := Int" } EQ_Contact(in1 := "BUFFER".PROCESS, in2 := 840)
      I_Contact( "ERROR" )
      I_Contact( "CYCLE PAUSE" )
   END_RUNG wire#w1
   RUNG wire#powerrail
      { S7_Templates := "SrcType := Int" } EQ_Contact(in1 := "BUFFER"."MODE SELECTION", in2 := 1)
      { S7_Templates := "SrcType := Int" } EQ_Contact(in1 := "BUFFER".PROCESS, in2 := 840)
      I_Contact( "IN".LSW_FWD_PUMP )
      Contact( "PW TANK_DRAIN".DONE )
      { S7_Templates := "time_type := Time" } "IEC_Timer_0_DB_135".TP(pt := T#1S, et =>)
      Move(in := 850, out1 => "BUFFER".PROCESS)
   END_RUNG
   RUNG wire#powerrail
      { S7_Templates := "SrcType := Int" } EQ_Contact(in1 := "BUFFER".PROCESS, in2 := 850)
      wire#w2
      R_Coil( "PW TANK_DRAIN".DONE )
   END_RUNG
   RUNG wire#powerrail
      { S7_Templates := "SrcType := Int" } EQ_Contact(in1 := "BUFFER"."MODE SELECTION", in2 := 0)
   END_RUNG wire#w2
   RUNG wire#powerrail
      { S7_Templates := "SrcType := Int" } EQ_Contact(in1 := "BUFFER".PROCESS, in2 := 0)
      wire#w3
      Coil( "PW TANK_DRAIN".RESET )
   END_RUNG
   RUNG wire#powerrail
      { S7_Templates := "SrcType := Int" } EQ_Contact(in1 := "BUFFER"."MODE SELECTION", in2 := 0)
   END_RUNG wire#w3
   // the same network as SCL:
   IF "AlwaysTRUE" THEN
       "PW TANK_DRAIN"("SET TIME" := "SET_PARAMETERS"."PW TANK_DRAIN_TIME_SV",   // "TIMING_BLOCK"
                       RESET := "PW TANK_DRAIN".RESET,
                       INPUT := "AlwaysTRUE" AND ("BUFFER"."MODE SELECTION" = 1) AND ("BUFFER".PROCESS = 840) AND NOT "ERROR" AND NOT "CYCLE PAUSE",
                       "PRESENT VALUE OF TIME" => "SET_PARAMETERS"."PW TANK_DRAIN_TIME_PV",
                       DONE => "PW TANK_DRAIN".DONE);
   END_IF;
   "IEC_Timer_0_DB_135".TP(IN := ("BUFFER"."MODE SELECTION" = 1) AND ("BUFFER".PROCESS = 840) AND NOT "IN".LSW_FWD_PUMP AND "PW TANK_DRAIN".DONE,
                           PT := T#1S);
   IF "IEC_Timer_0_DB_135".Q THEN "BUFFER".PROCESS := 850; END_IF;
   IF ("BUFFER".PROCESS = 850) OR ("BUFFER"."MODE SELECTION" = 0) THEN "PW TANK_DRAIN".DONE := FALSE; END_IF;
   "PW TANK_DRAIN".RESET := ("BUFFER".PROCESS = 0) OR ("BUFFER"."MODE SELECTION" = 0);
END_REGION

REGION Network 85: PW TANK_PUMP_CHASING_TIME(PBFV-12,PBFV13) FAKE TYPE AUDIT NOT OPERATE OUTPUT
